FUNCTION_BLOCK "GCS7_M_Flift1Airlock"	// FB 66
TITLE = Fluidlift Blower with 1 Airlock
//  
//COPYRIGHT:    (C) 1997  BUHLER AG, CH-9240 UZWIL, SWITZERLAND
//
//PRODUCT:      GCS7
//
//TITLE:        FB 66 Machine Control:Fluidlift with 1 Airlock 
//              Blower, Blow off valve and Airlock
//
//-------------------------------------------------------------------------
//
//IDENT:        AUTHOR:             DEPT:                       DATE:
//
//FB66.4.2      A. Egli             CT3                         24-Nov-2004
//              Starting condition Airlock: Pressure.StMinP 
//FB66.4.1      A. Egli             CT3                         18-Aug-2003
//              No blow off, when Blower is started in manual mode 
//FB66.4.0      A. Egli             CT3                         17-Jun-2002
//              New Release with one block 
//FB66.3.4      A.Egli              CT3                         18-Mar-2002
//              Pressure.InLocal moved to segment "Global End"
//FB66.3.3      S. Kalberer         CT3                         23-Oct-2000
//              Blower stopped: Do not open BlowOff valve
//FB66.3.2      A. Egli             CT3                         25-Mai-2000
//              InNoWaitMinP 
//FB66.3.1      A. Egli             CT3                         2-Mai-2000
//              InMonMinP moved from segment "Interlocking" to "Gloabl End"
//FB66.3.0      A. Egli             CT3                         11-Oct-1999
//              Local data reduced
//FB66.2C       A. Egli             CT3                         27-Aug-1999
//              Interlocking Airlock with InEnable 
//FB66.2B       K. Tischer          MU664                       06-Mrz-1999
//              CC FC2 not UC FC2
//FB66.2A       A. Egli             CT3                         04-Mai-1998
//              StFault = StCode 32
//FB66.1A       A.Egli              AEE61                       5-Jul-1997
//              1st Release in S7
//
//-------------------------------------------------------------------------
//
//PURPOSE:      MANUAL : see [LL.FL1xxMAN]
//
//RESTRICTIONS: S7
//              ACCU2: Pointer to dynamic datas of the machine
//              ACCU1: Pointer to parameter datas of the machine
//
//-------------------------------------------------------------------------
//
AUTHOR : EA
FAMILY : GCS7LL
NAME : Fluid1
VERSION : 4.2
VAR
  Ma : UDT 20660;
  Pressure : FB 16;	//Element
  BlowOff : FB 13;	//Element
  Blower : FB 12;	//Element
  Airlock : FB 12;	//Element
  HLInlet : FB 14;	//Element
END_VAR
VAR_TEMP
  tmpFaultStop : BOOL ;
  tmpFaultSum : BOOL ;
  tmpBlowerStopped : BOOL ;
  tmpBlowerStarted : BOOL ;
  tmpBlowOffStLN : BOOL ;
  tmpLenDyn : INT ;
END_VAR
BEGIN
NETWORK
TITLE =
      L     18;
      T     #tmpLenDyn;
NETWORK
TITLE = PC Control
//=== Test Object number =====================
      L     "SYS_DirectCtrlDB".PC.ObjectNo;	//PCControl.ObjectNo
      L     #Ma.Par.ParObjectNo;	//Input ObjectNo
      <>I;
      JC    aEnd;
//=== Test OType      ========================
      L     2066;	//Input object type
      L     "SYS_DirectCtrlDB".PC.ObjectType;	//PCControl.ObjectType
      <>I;
      JC    aEnd;
//=== Test Handshake =========================
      A     "SYS_DirectCtrlDB".PC.Hsk.FExamine;	// Handshake.FExamine
      JC    aExa;
      A     "SYS_DirectCtrlDB".PC.Hsk.FDefineCmd;	// Handshake.FDefineCmd
      JC    aCmd;
      A     "SYS_DirectCtrlDB".PC.Hsk.FDefinePara;	// Handshake.FDefinePara
      JC    pPar;
aIni: L     2;	// FcInit
      UC    "SYS_DirectCtrl";
      JU    aEnd;
// Write parameter 
pPar: LAR1  P#DBX 58.0;
      L     P#6.0;
      +AR1;
      L     DBW [AR1,P#4.0];
      T     #Ma.Par.ParClearingTime;
// Write new commands from PC to Interface of group 
aCmd: A     "SYS_DirectCtrlDB".PC.Cmd1[8];	//Cmd1[8]=CmdOff
      S     #Ma.CmdOff;
      A     "SYS_DirectCtrlDB".PC.Cmd1[9];	//Cmd1[9]=CmdOn
      S     #Ma.CmdOn;
      A     "SYS_DirectCtrlDB".PC.Cmd1[10];	//Cmd1[10]=CmdNext
      S     #Ma.CmdNext;
      A     "SYS_DirectCtrlDB".PC.Cmd1[11];	//Cmd1[11]=CmdFaultReset
      S     #Ma.CmdFaultReset;
      A     "SYS_DirectCtrlDB".PC.Cmd1[13];	//Cmd1[13]=CmdManualOn
      S     #Ma.InManual;
      A     "SYS_DirectCtrlDB".PC.Cmd2[13];	//Cmd2[13]=CmdManualOff
      R     #Ma.InManual;
      A     "SYS_DirectCtrlDB".PC.Cmd1[14];	//Cmd1[14]=CmdManualOn
      S     #Ma.CmdAirlockOff;
      A     "SYS_DirectCtrlDB".PC.Cmd1[6];	//Cmd1[6]=CmdClearingOn
      S     #Ma.InClearing;
      A     "SYS_DirectCtrlDB".PC.Cmd2[6];	//Cmd2[6]=CmdClearingOff
      R     #Ma.InClearing;
      JU    aIni;
aExa: TAR2;	// Address Dynamic datas
      T     "SYS_DirectCtrlDB".GC.InDynAddr;	// -->PCControl.GC.InDynAddr
      L     #tmpLenDyn;	// Length Dynamic datas
      T     "SYS_DirectCtrlDB".GC.InDynLen;	// -->PCControl.GC.InDynLen
      L     0;
      T     "SYS_DirectCtrlDB".GC.InParaAddr;	// -->PCControl.GC.InParaAddr
      T     "SYS_DirectCtrlDB".GC.InParaLen;	// -->PCControl.GC.InParaLen
      L     1;	// Code FcExamine
      UC    "SYS_DirectCtrl";
      L     10;	//Revision
      T     "SYS_DirectCtrlDB".GC.Revision;
aEnd: NOP   0;
NETWORK
TITLE = Interlocking
//===Dynamic Group Orders===
      A     "GCS7_Gr_OutManualOn";	//Gr.OutManualOn
      S     #Ma.InManual;
      A     "GCS7_Gr_OutManualOff";	//Gr.OutManualOff
      R     #Ma.InManual;
      A     #Ma.InManual;
      S     "GCS7_Gr_InManual";	//Gr.InManual
//--- Fault----
      A     #Pressure.StFault;
      O     #BlowOff.StFault;
      O     #Blower.StFault;
      O     #Airlock.StFault;
      O     #HLInlet.StFault;
      =     #tmpFaultSum;
//Temporare signal
      A     #BlowOff.StLN;
      =     #tmpBlowOffStLN;
      A     #Ma.Par.ParBlowerExternal;
      A     #Ma.InBlowerStarted;
      O;
      AN    #Ma.Par.ParBlowerExternal;
      A     #Blower.StStartedFwd;
      =     #tmpBlowerStarted;
      A     #Ma.Par.ParBlowerExternal;
      AN    #Ma.InBlowerStarted;
      O;
      AN    #Ma.Par.ParBlowerExternal;
      A     #Blower.StStopped;
      =     #tmpBlowerStopped;
//--- Interlocking blow off
      A     #Ma.InClearing;
      A     #Ma.StCleared;
//[3.3]   ON    #tmpBlowerStarted;
      O     #Ma.InBlowOff;
      AN    #Blower.InManual;	//[4.1]
      =     #BlowOff.InEnableHN;
      AN    #BlowOff.InEnableHN;
      =     #BlowOff.InEnableLN;
//[->3.3  U     #Ma.CmdNext; 
//        UN    #Ma.InManual;
//        O     #Ma.CmdOn;
//        O     #tmpBlowerStarted;
      SET;	//<-3.3]
      S     #BlowOff.CmdNext;
// 
//--- Interlocking blower
      AN    #Pressure.StOverP;
      AN    #Pressure.StFault;
      =     #Ma.OutEnableBlower;
      AN    #Pressure.StOverP;
      AN    #Pressure.StFault;
      A     #Ma.InEnable;
      AN    #BlowOff.StFault;
      AN    #Ma.CmdOff;
      =     #Blower.InEnableFwd;
// 
//[3.3]   U     #BlowOff.StHN;
//[3.3]   ON    #Ma.Par.ParWithBlowOff;
//[3.3]   U(;
      A     #Ma.CmdNext;
      AN    #Ma.InManual;
      O     #Ma.CmdOn;
//[3.3]   ); 
      S     #Blower.CmdNext;
// 
      A     #Ma.InSeqStop;
      =     #Blower.InSeqStop;
// 
//--- Interlocking airlock 
      A     #BlowOff.StLN;
      ON    #Ma.Par.ParWithBlowOff;
      A     #tmpBlowerStarted;
      A     #Ma.InEnable;	// [Rel 2C]
      AN    #Ma.InClearing;
      AN    #Ma.InBlowOff;
      AN    #Pressure.StOverP;
      AN    #Pressure.StCtoOverP;
      AN    #Pressure.StFault;
      AN    #Ma.CmdOff;
      AN    #Ma.CmdAirlockOff;
      =     #Airlock.InEnableFwd;
// 
      A     #Ma.CmdNext;
      AN    #Ma.InManual;
      O     #Ma.CmdOn;
      A(;	//[4.2]
      A     #Pressure.StMinP;	//[4.2]
      O     #Ma.InNoWaitMinP;	//[4.2]
      );	//[4.2]
      S     #Airlock.CmdNext;
// 
      A     #Ma.InSeqStop;
      =     #Airlock.InSeqStop;
// 
//--- Local mode --
      A     #Ma.InLocal;
      AN    #Ma.InManual;
      =     #Blower.InLocal;
      =     #Airlock.InLocal;
      =     #HLInlet.InLocal;
      A     #Ma.InLocal;
      AN    #Ma.InManual;
      A     #tmpBlowerStopped;
      =     #BlowOff.InLocal;
//      =     #Pressure.InLocal //[3.4]
//--- Fault Reset -------------
      A     #Ma.CmdFaultReset;
      S     #Pressure.CmdFaultReset;
      S     #BlowOff.CmdFaultReset;
      S     #Blower.CmdFaultReset;
      S     #Airlock.CmdFaultReset;
      S     #HLInlet.CmdFaultReset;
//Warning
      A     #Pressure.OutNoMinP;
      =     #Ma.OutWarning;
NETWORK
TITLE = Call PRange: Pressure
      CALL  #Pressure;
NETWORK
TITLE = Call VLS: Blow off
      AN    #Ma.Par.ParWithBlowOff;
      JC    el3;
      CALL  #BlowOff;
NETWORK
TITLE = Call Blower
el3:  A     #Ma.Par.ParBlowerExternal;
      JC    el4;
      CALL  #Blower;
NETWORK
TITLE = Call Airlock
el4:  CALL  #Airlock;
NETWORK
TITLE = Call Digital Input: HLInlet
      AN    #Ma.Par.ParWithHLInlet;
      JC    StJ0;
      CALL  #HLInlet;
NETWORK
TITLE = Jump to actual state
StJ0: A     #Ma.StStopped;
      JC    S0;	// ===> State
      A     #Ma.StStarted;
      JC    S2;	// ===> State
      A     #Ma.StStarting;
      JC    S1;	// ===> State
      A     #Ma.StStopping;
      JC    S3;	// ===> State
      A     #Ma.StClearing;
      JC    S5;	// ===> State
      A     #Ma.StCleared;
      JC    S6;	// ===> State
      A     #Ma.StFault;
      JC    S4;	// ===> State
NETWORK
TITLE = Stopped
//any Transition 
xxS0: S     #Ma.StStopped;	// ===> Initialisation
//=== Logic
// Condition for StFault
S0:   A     #tmpFaultSum;
      R     #Ma.StStopped;
      JC    xxS4;	//--> StFault
// Condition for StStarting
      AN    #tmpBlowerStopped;
      ON    #Airlock.StStopped;
      R     #Ma.StStopped;
      JC    xxS1;	//--> StStarting
      JU    OUT;
NETWORK
TITLE = StStarting
//any Transition 
xxS1: S     #Ma.StStarting;
      JU    OUT;
//=== Logic
// Condition for StFault
S1:   A     #tmpFaultSum;
      R     #Ma.StStarting;
      JC    xxS4;	//--> StFault
// Condition for StStopping
      AN    #Blower.StStarting;
      AN    #Blower.StStartedFwd;
      AN    #tmpBlowerStarted;
      R     #Ma.StStarting;
      JC    xxS3;	//-->StStopping
// Condition for StStarted
      A     #BlowOff.StLN;
      ON    #Ma.Par.ParWithBlowOff;
      A     #tmpBlowerStarted;
      A     #Airlock.StStartedFwd;
      R     #Ma.StStarting;
      JC    xxS2;	//-->StStarted
// Condition for StClearing
      AN    #Ma.Par.ParWithBlowOff;
      O     #tmpBlowOffStLN;
      A     #tmpBlowerStarted;
      AN    #Airlock.StStarting;
      R     #Ma.StStarting;
      JC    xxS5;	//-->StClearing
      JU    OUT;
NETWORK
TITLE = StStarted
//any Transition 
xxS2: S     #Ma.StStarted;
//=== Logic
// Condition for StFault
S2:   A     #tmpFaultSum;
      R     #Ma.StStarted;
      JC    xxS4;	//--> StFault
// Condition for StClearing
      AN    #Airlock.StStartedFwd;
      R     #Ma.StStarted;
      JC    xxS5;	//-->StClearing  
// Condition for StStarted
      ON    #tmpBlowerStarted;
      R     #Ma.StStarted;
      JC    xxS3;	//-->StStopping
      JU    OUT;
NETWORK
TITLE = Stopping
//any Transition 
xxS3: S     #Ma.StStopping;
      JU    OUT;
//=== Logic
// Condition for StFault
S3:   A     #tmpFaultSum;
      R     #Ma.StStopping;
      JC    xxS4;	//--> StFault
// Condition for StStopped
      A     #tmpBlowerStopped;
      A     #Airlock.StStopped;
      R     #Ma.StStopping;
      JC    xxS0;	//-->StStopped
// Condition for StStarting
      AN    #Blower.StStopping;
      AN    #Ma.Par.ParBlowerExternal;
      O     #tmpBlowerStarted;
      AN    #Airlock.StStopping;
      R     #Ma.StStopping;
      JC    xxS1;	//-->StStarting
      JU    OUT;
NETWORK
TITLE = Fault
//any Transition 
xxS4: S     #Ma.StFault;
      JU    OUT;
//=== Logic
S4:   A     #tmpFaultSum;
      JC    OUT;
//    ---- Transition --
      R     #Ma.StFault;
      JU    xxS0;	//-->StStopping 
NETWORK
TITLE = StClearing
//any Transition 
xxS5: S     #Ma.StClearing;
S5J2: L     #Ma.Par.ParClearingTime;
      T     #Ma.Par.OutClearingTime;
      JU    OUT;
//=== Logic
// Condition for StFault
S5:   A     #tmpFaultSum;
      R     #Ma.StClearing;
      JC    xxS4;	//-->StFault
// Condition for StStopping
      AN    #tmpBlowerStarted;
      R     #Ma.StClearing;
      JC    xxS3;	//-->StStopping  
// Condition for StStarted
      A     #tmpBlowerStarted;
      A     #Airlock.StStartedFwd;
      R     #Ma.StClearing;
      JC    xxS2;	//-->StStarted
// Condition for StCleared
      L     0;
      L     #Ma.Par.OutClearingTime;
      >=I;
      A(;
      A     #Pressure.StMinP;
      O     #Ma.InNoWaitMinP;	// [3.2]
      );
      R     #Ma.StClearing;
      JC    xxS6;	//-->StCleared 
      AN    #BlowOff.StLN;
      A     #Ma.Par.ParWithBlowOff;
      O;
      AN    #Pressure.StMinP;
      AN    #Ma.InNoWaitMinP;	// [3.2]
      JC    S5J2;
      ON    "GCS7_Gr_OutTick500ms";	//Gr.OutTick500ms
      JC    OUT;
      +     -5;
      T     #Ma.Par.OutClearingTime;
      JU    OUT;
NETWORK
TITLE = StCleared
//any Transition 
xxS6: S     #Ma.StCleared;
      JU    OUT;
//=== Logic
// Condition for StFault
S6:   A     #tmpFaultSum;
      R     #Ma.StCleared;
      JC    xxS4;	//-->StFault
// Condition for StStopping
      AN    #tmpBlowerStarted;
      R     #Ma.StCleared;
      JC    xxS3;	//-->StStopping
// Condition for StStarted
      A     #tmpBlowerStarted;
      A     #Airlock.StStartedFwd;
      R     #Ma.StCleared;
      JC    xxS2;	//-->StStarted
      JU    OUT;
NETWORK
TITLE = State Code
// State     StCode
// ----------------------
// StFault 32
// StStopped          1
// StStarting         2
// StStarted          3
// StClearing         4
// StCleared          5
// StClearingWarning  6
// StStopping         7
OUT:  A     #Ma.StStopped;
      L     1;	//Code=StStopped
      JC    Code;
      A     #Ma.StStarted;
      L     3;	//Code=StStarted
      JC    Code;
      A     #Ma.StCleared;
      L     5;	//Code=StCleared
      JC    Code;
      A     #Ma.StClearing;
      AN    #Ma.OutWarning;
      L     4;	//Code=StClearing 
      JC    Code;
      A     #Ma.StClearing;
      L     6;	//Code=StWarning 
      JC    Code;
      A     #Ma.StStarting;
      L     2;	//Code=StStarting
      JC    Code;
      A     #Ma.StStopping;
      L     7;	//Code=StStopping 
      JC    Code;
      L     32;	//Code=StFault 
Code: L     #Ma.StCode;	// Old state code
      TAK;
      T     #Ma.StCode;	// Save state code
      <>I;
      L     3;
      CC    "SYS_CBitCtrl";	//Set change bit
NETWORK
TITLE = Global End
      CLR;	//---Clear all commands
      =     #Ma.CmdOn;
      =     #Ma.CmdOff;
      =     #Ma.CmdNext;
      =     #Ma.CmdFaultReset;
      =     #Ma.CmdAirlockOff;
// 
//--- Interlocking pressure 
      A     #BlowOff.StLN;
      ON    #Ma.Par.ParWithBlowOff;
      AN    #Airlock.StStartedFwd;
      A     #tmpBlowerStarted;
      =     #Pressure.InMonMinP;
// 
//--- Local mode --       
      A     #BlowOff.InLocal;	//[3.4]
      =     #Pressure.InLocal;	//[3.4]
// 
//--- Interlocking HL 
      SET;
      =     #HLInlet.InMonFalse;
END_FUNCTION_BLOCK

FUNCTION_BLOCK "GCS7_M_Flift2Airlock"	// FB 67
TITLE = Fluidlift Blower with 2 Airlock
//  
//COPYRIGHT:    (C) 1997  BUHLER AG, CH-9240 UZWIL, SWITZERLAND
//
//PRODUCT:      GCS7
//
//TITLE:        FB 67 Machine Control:Fluidlift 2 Airlock and 2 Shutoff Valve
//              Blower, Blow off valve and Airlock
//
//-------------------------------------------------------------------------
//
//IDENT:        AUTHOR:             DEPT:                       DATE:
//
//FB67.6.7      A. Egli             BASE                        10-Apr-2008
//              StStarting -> StStopping ParExternal
//FB67.6.6      A. Egli             CT3                         04-Mar-2005
//              Support continuous valve for ShutOff and BlowOff 
//FB67.6.5      A. Egli             CT3                         04-Mar-2005
//              Start Blower before opening ShutOffA or ShutOffB 
//FB67.6.4      A. Egli             CT3                         20-Sep-2004
//              Interlocking Subtype Diverter without BlowOff valve
//FB67.6.3      A. Egli             CT3                         10-Jun-2004
//              Diverter.InLocal
//FB67.6.2      A. Egli             CT3                         19-Sep-2003
//              InMonFalse mode to global end function
//FB67.6.1      A. Egli             CT3                         18-Aug-2003
//              No blow off, when Blower is started in manual mode 
//FB67.6.0      A. Egli             CT3                         17-Jun-2002
//              New Release with one block 
//FB67.5.7      A.Egli              CT3                         18-Mar-2002
//              Pressure.InLocal moved to segment "Global End"
//FB67.5.6      A.Egli              CT3                         29-Oct-2001
//              InLocal of HL moved to segment "Global End"
//FB67.5.5      A.Egli              CT3                         16-May-2001
//              - Close Valve with InSeqStop
//              - Monitoring only active HLInlet  
//FB67.5.4      Ph.Engler           MU664                       15-May-2001
//              - Diverter.CmdFaultReset corrected
//FB67.5.3      Ph.Engler           MU664                       08-Jan-2000
//              InBlowOff without a blowoff valve closes directly
//              the ShutOffA valve.
//FB67.5.2      Ph.Engler           MU664                       29-Dec-2000
//              - Enable airlock A on a single line type and shutt off valve
//              - OutEnableBlower implemented
//              - InMonMinP moved from segment "Interlocking" to "Gloabl End"
//FB67.5.1      S. Kalberer         CT3                         23-Oct-2000
//              Blower stopped: Do not open BlowOff valve
//FB67.5.0      A. Egli             CT3                    20-Sep-2000
//              With Diverter valve
//FB67.4.0      A. Egli             CT3                    26-Mai-2000
//              Single line with ShutOff valves
//              InNoWaitMinP 
//FB67.3.1      A. Egli             CT3                    28-Jan-2000
//              Interlocking blower
//FB67.3.0      A. Egli             CT3                         11-Oct-1999
//              Local data reduced
//FB67.2B       K. Tischer          MU664                       06-Mrz-1999
//              CC FC2 not UC FC2
//FB67.2A       A. Egli             CT3                         04-Mai-1998
//              StFault = StCode 32
//FB67.1A       A. Egli              AEE61                      27-Nov-1997
//              1st Release in S7
//
//-------------------------------------------------------------------------
//
//PURPOSE:      MANUAL : see [LL.FL2xxMAN]
//
//RESTRICTIONS: S7
//              ACCU2: Pointer to dynamic datas of the machine
//              ACCU1: Pointer to parameter datas of the machine
//
//-------------------------------------------------------------------------
//
AUTHOR : EA
FAMILY : GCS7LL
NAME : Fluid2AV
VERSION : 6.6
VAR
  Ma : UDT 20670;
  Pressure : FB 16;	//Element
  BlowOff : FB 13;	//Element
  Blower : FB 12;	//Element
  ShutOffA : FB 13;	//Element
  ShutOffB : FB 13;	//Element
  AirlockA : FB 12;	//Element
  AirlockB : FB 12;	//Element
  HLInletA : FB 14;	//Element
  HLInletB : FB 14;	//Element
  Diverter : FB 13;	//Element
END_VAR
VAR_TEMP
  tmpFaultStop : BOOL ;
  tmpFaultSum : BOOL ;
  tmpEnable : BOOL ;
  tmpEnableAirlock : BOOL ;
  tmpNext : BOOL ;
  tmpBlowOff : BOOL ;
  tmpBlowerStopped : BOOL ;
  tmpBlowerStarted : BOOL ;
  tmpBlowOffStLN : BOOL ;
  tmpWayA : BOOL ;
  tmpWayB : BOOL ;
  tmpWithShutOffValves : BOOL ;
  tmpWithDiverterValves : BOOL ;
  tmpWayAOK : BOOL ;
  tmpWayBOK : BOOL ;
  tmpCloseValve : BOOL ;
  tmpPressureLocal : BOOL ;
  tmpLenDyn : INT ;
END_VAR
BEGIN
NETWORK
TITLE =
      L     18;
      T     #tmpLenDyn;
NETWORK
TITLE = PC Control
//=== Test Object number =====================
      L     "SYS_DirectCtrlDB".PC.ObjectNo;	//PCControl.ObjectNo
      L     #Ma.Par.ParObjectNo;	//Input ObjectNo
      <>I;
      JC    aEnd;
//=== Test OType  ========================
      L     2067;	//Input object type
      L     "SYS_DirectCtrlDB".PC.ObjectType;	//PCControl.ObjectType
      <>I;
      JC    aEnd;
//=== Test Handshake =========================
      A     "SYS_DirectCtrlDB".PC.Hsk.FExamine;	// Handshake.FExamine
      JC    aExa;
      A     "SYS_DirectCtrlDB".PC.Hsk.FDefineCmd;	// Handshake.FDefineCmd
      JC    aCmd;
      A     "SYS_DirectCtrlDB".PC.Hsk.FDefinePara;	// Handshake.FDefinePara
      JC    pPar;
aIni: L     2;	// FcInit
      UC    "SYS_DirectCtrl";
      JU    aEnd;
// Write parameter 
pPar: LAR1  P#DBX 58.0;
      L     P#6.0;
      +AR1;
      L     DBW [AR1,P#4.0];
      T     #Ma.Par.ParClearingTime;
// Write new commands from PC to Interface of group 
aCmd: A     "SYS_DirectCtrlDB".PC.Cmd1[8];	//Cmd1[8]=CmdOff
      S     #Ma.CmdOff;
      A     "SYS_DirectCtrlDB".PC.Cmd1[9];	//Cmd1[9]=CmdOn
      S     #Ma.CmdOn;
      A     "SYS_DirectCtrlDB".PC.Cmd1[10];	//Cmd1[10]=CmdNext
      S     #Ma.CmdNext;
      A     "SYS_DirectCtrlDB".PC.Cmd1[11];	//Cmd1[11]=CmdFaultReset
      S     #Ma.CmdFaultReset;
      A     "SYS_DirectCtrlDB".PC.Cmd1[13];	//Cmd1[13]=CmdManualOn
      S     #Ma.InManual;
      A     "SYS_DirectCtrlDB".PC.Cmd2[13];	//Cmd2[13]=CmdManualOff
      R     #Ma.InManual;
      A     "SYS_DirectCtrlDB".PC.Cmd1[14];	//Cmd1[14]=CmdManualOn
      S     #Ma.CmdAirlockOff;
      A     "SYS_DirectCtrlDB".PC.Cmd1[1];	//Cmd1[1]=CmdWayA
      R     #Ma.InWayB;
      A     "SYS_DirectCtrlDB".PC.Cmd2[1];	//Cmd2[2]=CmdWayB
      S     #Ma.InWayB;
      A     "SYS_DirectCtrlDB".PC.Cmd1[6];	//Cmd1[6]=CmdClearingOn
      S     #Ma.InClearing;
      A     "SYS_DirectCtrlDB".PC.Cmd2[6];	//Cmd2[6]=CmdClearingOff
      R     #Ma.InClearing;
      JU    aIni;
aExa: TAR2;	// Address Dynamic datas
      T     "SYS_DirectCtrlDB".GC.InDynAddr;	// -->PCControl.GC.InDynAddr
      L     #tmpLenDyn;	// Length Dynamic datas
      T     "SYS_DirectCtrlDB".GC.InDynLen;	// -->PCControl.GC.InDynLen
      L     0;
      T     "SYS_DirectCtrlDB".GC.InParaAddr;	// -->PCControl.GC.InParaAddr
      T     "SYS_DirectCtrlDB".GC.InParaLen;	// -->PCControl.GC.InParaLen
      L     1;	// Code FcExamine
      UC    "SYS_DirectCtrl";
      L     10;	//Revision
      T     "SYS_DirectCtrlDB".GC.Revision;
aEnd: NOP   0;
NETWORK
TITLE = Interlocking
//===Dynamic Group Orders===
      A     "GCS7_Gr_OutManualOn";	//Gr.OutManualOn
      S     #Ma.InManual;
      A     "GCS7_Gr_OutManualOff";	//Gr.OutManualOff
      R     #Ma.InManual;
      A     #Ma.InManual;
      S     "GCS7_Gr_InManual";	//Gr.InManual
      A     #Ma.InManual;
      ON    #Ma.InLocal;
      A     #Ma.InEnable;
      AN    #Ma.CmdOff;
      =     #tmpEnable;
//Temporare signal
      AN    #Ma.InWayB;
      O     #Ma.InWayAB;
      =     #tmpWayA;
      A     #Ma.InWayB;
      O     #Ma.InWayAB;
      =     #tmpWayB;
      A     #BlowOff.StLN;
      =     #tmpBlowOffStLN;
      A     #Ma.Par.ParWithShutOffValves;
      ON    #Ma.Par.ParSingleLine;
      =     #tmpWithShutOffValves;
      A     #Ma.Par.ParBlowerExternal;
      A     #Ma.InBlowerStarted;
      O;
      AN    #Ma.Par.ParBlowerExternal;
      A     #Blower.StStartedFwd;
      =     #tmpBlowerStarted;
      A     #Ma.Par.ParBlowerExternal;
      AN    #Ma.InBlowerStarted;
      O;
      AN    #Ma.Par.ParBlowerExternal;
      A     #Blower.StStopped;
      =     #tmpBlowerStopped;
      A     #Ma.InSeqStop;	//[5.5]
      O     #Ma.InLocal;	//[5.5]
      AN    #Ma.InManual;	//[5.5]
      A     #tmpBlowerStopped;	//[5.5]
      AN    #Blower.InManual;	//[6.1]
      =     #tmpCloseValve;	//[5.5]
//--- Fault----
      A     #Diverter.StFault;
      A     #Ma.Par.ParWithDiverter;
      O     #Pressure.StFault;
      O     #BlowOff.StFault;
      O     #ShutOffA.StFault;
      O     #ShutOffB.StFault;
      O     #Blower.StFault;
      O     #AirlockA.StFault;
      O     #AirlockB.StFault;
      O     #HLInletA.StFault;
      O     #HLInletB.StFault;
      =     #tmpFaultSum;
//CmdNext
      A     #Ma.CmdNext;
      AN    #Ma.InManual;
      O     #Ma.CmdOn;
      =     #tmpNext;
//[5.1]   U       #BlowOff.StHN;
//[5.1]   ON      #Ma.Par.ParWithBlowOff;
      A     #tmpNext;
      S     #Blower.CmdNext;
      A     #tmpNext;
      S     #Blower.CmdNext;
      S     #AirlockA.CmdNext;
      S     #AirlockB.CmdNext;
      SET;
      S     #BlowOff.CmdNext;
      A(;	//[6.5]
      A     #tmpBlowerStarted;	//[6.5]
      ON    #Ma.Par.ParWithBlowOff;	//[6.5]
      );	//[6.5]
      O;
      A     #ShutOffA.InEnableLN;	//[6.5]
      AN    #ShutOffA.StLN;	//[6.5]
      S     #ShutOffA.CmdNext;
      A(;	//[6.5]
      A     #tmpBlowerStarted;	//[6.5]
      ON    #Ma.Par.ParWithBlowOff;	//[6.5]
      );	//[6.5]
      O(;
      A     #ShutOffB.InEnableLN;	//[6.5]
      AN    #ShutOffB.StLN;	//[6.5]
      );
      S     #ShutOffB.CmdNext;
      AN    #Ma.Par.ParWithDiverter;
      JC    InX1;
      S     #Diverter.CmdNext;
//--- Interlocking blow off
InX1: A     #Diverter.StLN;
      ON    #Ma.Par.ParWithDiverter;
      A     #ShutOffA.StHN;
      A(;
      A     #tmpWayA;
      O     #Ma.Par.ParSingleLine;
      );
      =     #tmpWayAOK;
      A     #Diverter.StHN;
      ON    #Ma.Par.ParWithDiverter;
      A     #ShutOffB.StHN;
      A     #tmpWayB;
      AN    #Ma.Par.ParSingleLine;
      =     #tmpWayBOK;
      A     #Ma.InClearing;
      A     #Ma.StCleared;
//[5.1]   ON      #tmpBlowerStarted;
      O     #Ma.InBlowOff;
      A     #Ma.Par.ParWithBlowOff;
      =     #tmpBlowOff;
      AN    #tmpWayAOK;
      AN    #tmpWayBOK;
      A     #tmpWithShutOffValves;
      O     #tmpBlowOff;
      AN    #tmpCloseValve;	//[5.5]
      =     #BlowOff.InEnableHN;
      AN    #BlowOff.InEnableHN;
      =     #BlowOff.InEnableLN;
//--- Interlocking ShutOff Valve
      A     #Diverter.StHN;	//[6.4]
      ON    #Ma.Par.ParWithDiverter;	//[6.4]
      A     #ShutOffB.StHN;
      A     #tmpWayB;
      AN    #tmpWayA;
      O;
      A     #tmpBlowOff;
      A     #BlowOff.StHN;
      O;
      A     #Ma.InBlowOff;
      AN    #Ma.Par.ParWithBlowOff;
      O;
      A     #BlowOff.StHN;
      A     #tmpWayB;
      A     #Ma.Par.ParWithDiverter;
      O     #tmpCloseValve;	//[5.5]
      =     #ShutOffA.InEnableLN;
      R     #ShutOffA.InEnableHN;	//[6.6]
      A     #tmpWayA;
      O     #Ma.Par.ParSingleLine;
      AN    #ShutOffA.InEnableLN;
      A(;
      A     #ShutOffB.StHN;	//[6.4]
      AN    #Ma.Par.ParWithBlowOff;	//[6.4]
      O     #Diverter.StLN;
      ON    #Ma.Par.ParWithDiverter;
      );
      S     #ShutOffA.InEnableHN;	//[6.6]
      R     #ShutOffA.InEnableLN;	//[6.6]
      A     #Diverter.StLN;	//[6.4]
      ON    #Ma.Par.ParWithDiverter;	//[6.4]
      A     #ShutOffA.StHN;
      A     #tmpWayA;
      AN    #tmpWayB;
      O;
      A     #tmpBlowOff;
      A     #BlowOff.StHN;
      O;
      A     #BlowOff.StHN;
      A     #tmpWayA;
      A     #Ma.Par.ParWithDiverter;
      O     #tmpCloseValve;	//[5.5]
      =     #ShutOffB.InEnableLN;
      R     #ShutOffB.InEnableHN;	//[6.6]
      AN    #ShutOffB.InEnableLN;
      A     #tmpWayB;
      A(;
      A     #ShutOffA.StHN;	//[6.4]
      AN    #Ma.Par.ParWithBlowOff;	//[6.4]
      O     #Diverter.StHN;
      ON    #Ma.Par.ParWithDiverter;
      );
      S     #ShutOffB.InEnableHN;	//[6.6]
      R     #ShutOffB.InEnableLN;	//[6.6]
//--- Interlocking blower
      AN    #Pressure.StOverP;	//[5.2]
      AN    #Pressure.StFault;	//[5.2]
      =     #Ma.OutEnableBlower;	//[5.2]
      A     #BlowOff.StHN;
      A     #Ma.Par.ParWithBlowOff;
      O     #ShutOffA.StHN;	//[3.1]
      O     #ShutOffB.StHN;	//[3.1]
      ON    #tmpWithShutOffValves;	//[4.0]
      A     #tmpEnable;
      AN    #Pressure.StOverP;
      AN    #Pressure.StFault;
      AN    #BlowOff.StFault;
      =     #Blower.InEnableFwd;
// 
      A     #Ma.InSeqStop;
      AN    #Ma.InManual;	//[5.5]
      =     #Blower.InSeqStop;
// 
//--- Interlocking airlock 
      A     #BlowOff.StLN;
      ON    #Ma.Par.ParWithBlowOff;
      AN    #Ma.InClearing;
      A     #tmpEnable;
      A     #tmpBlowerStarted;
      AN    #Pressure.StOverP;
      AN    #Pressure.StCtoOverP;
      AN    #Pressure.StFault;
      AN    #Ma.CmdAirlockOff;
      AN    #Ma.InBlowOff;
      =     #tmpEnableAirlock;
      A     #ShutOffB.StLN;
      O     #tmpWayB;
      O     #Ma.Par.ParSingleLine;	//[5.2]
      A     #ShutOffA.StHN;
      ON    #tmpWithShutOffValves;
      A     #tmpEnableAirlock;
      A     #tmpWayA;
      AN    #Ma.InDisableAirlockA;
      A(;
      A     #Diverter.StLN;
      ON    #Ma.Par.ParWithDiverter;
      );
      =     #AirlockA.InEnableFwd;
      A     #ShutOffA.StLN;
      O     #tmpWayA;
      A     #ShutOffB.StHN;
      A     #tmpEnableAirlock;
      A     #tmpWayB;
      AN    #Ma.Par.ParSingleLine;
      O(;
      A     #ShutOffA.StHN;
      ON    #tmpWithShutOffValves;
      A     #tmpEnableAirlock;
      A     #tmpWayB;
      O     #AirlockA.InEnableFwd;
      A     #Ma.Par.ParSingleLine;
      );
      AN    #Ma.InDisableAirlockB;
      A(;
      A     #Diverter.StHN;
      ON    #Ma.Par.ParWithDiverter;
      );
      =     #AirlockB.InEnableFwd;
// 
      A     #Ma.InSeqStop;
      AN    #Ma.InManual;	//[5.5]
      =     #AirlockA.InSeqStop;
      =     #AirlockB.InSeqStop;
// 
//--- Interlocking pressure  [5.2] moved to "global end"
// 
//--- Interlocking HL        [6.2] moved to "global end"
//--- Interlocking Diverter
      AN    #Ma.Par.ParWithDiverter;
      JC    EnX1;
      A(;	//[6.4]
      A     #BlowOff.StHN;
      A     #ShutOffB.StLN;	//[6.4]
      A     #Ma.Par.ParWithBlowOff;	//[6.4]
      O;
      A     #ShutOffA.StHN;	//[6.4]
      AN    #Ma.Par.ParWithBlowOff;	//[6.4]
      O;
      A     #ShutOffB.StLN;	//[6.4]
      AN    #Ma.Par.ParWithBlowOff;	//[6.4]
      );	//[6.4]
      A     #tmpWayA;
      S     #Diverter.InEnableLN;
      R     #Diverter.InEnableHN;
      A(;	//[6.4]
      A     #BlowOff.StHN;
      A     #ShutOffA.StLN;	//[6.4]
      A     #Ma.Par.ParWithBlowOff;	//[6.4]
      O;
      A     #ShutOffB.StHN;	//[6.4]
      AN    #Ma.Par.ParWithBlowOff;	//[6.4]
      O;
      A     #ShutOffA.StLN;	//[6.4]
      AN    #Ma.Par.ParWithBlowOff;	//[6.4]
      );	//[6.4]
      A     #tmpWayB;
      R     #Diverter.InEnableLN;
      S     #Diverter.InEnableHN;
// 
//--- Local mode --
EnX1: A     #Ma.InLocal;
      AN    #Ma.InManual;
      =     #Blower.InLocal;
      =     #AirlockA.InLocal;
      =     #AirlockB.InLocal;
      =     #Diverter.InLocal;	//[6.3]
      A     #Ma.InLocal;
      AN    #Ma.InManual;
      A     #tmpBlowerStopped;
      =     #tmpPressureLocal;
      A     #BlowOff.StLN;	//[5.5]
      O     #BlowOff.StFault;	//[5.5]
      A     #tmpPressureLocal;	//[5.5]
      S     #BlowOff.InLocal;	//[5.5]
      A     #ShutOffA.StLN;	//[5.5]
      O     #ShutOffA.StFault;	//[5.5]
      A     #tmpPressureLocal;	//[5.5]
      S     #ShutOffA.InLocal;	//[5.5]
      A     #ShutOffB.StLN;	//[5.5]
      O     #ShutOffB.StFault;	//[5.5]
      A     #tmpPressureLocal;	//[5.5]
      S     #ShutOffB.InLocal;	//[5.5]
      AN    #tmpPressureLocal;	//[5.5]
      R     #BlowOff.InLocal;
      R     #ShutOffA.InLocal;
      R     #ShutOffB.InLocal;
//--- Fault Reset -------------
      A     #Ma.CmdFaultReset;
      S     #Pressure.CmdFaultReset;
      S     #BlowOff.CmdFaultReset;
      S     #ShutOffA.CmdFaultReset;
      S     #ShutOffB.CmdFaultReset;
      S     #Blower.CmdFaultReset;
      S     #AirlockA.CmdFaultReset;
      S     #AirlockB.CmdFaultReset;
      S     #HLInletA.CmdFaultReset;
      S     #HLInletB.CmdFaultReset;
      AN    #Ma.Par.ParWithDiverter;
      JC    FrX1;
      A     #Ma.CmdFaultReset;	// [5.4]
      S     #Diverter.CmdFaultReset;
//Warning
FrX1: A     #Pressure.OutNoMinP;
      =     #Ma.OutWarning;
NETWORK
TITLE = Call PRange: Pressure
      CALL  #Pressure;
NETWORK
TITLE = Call VLS: Blow off
      AN    #Ma.Par.ParWithBlowOff;
      JC    el3;
      CALL  #BlowOff;
NETWORK
TITLE = Call VLS: ShutOffA
el3:  AN    #tmpWithShutOffValves;
      JC    el4;
      CALL  #ShutOffA;
NETWORK
TITLE = Call VLS: ShutOffB
el4:  A     #Ma.Par.ParSingleLine;
      JC    el5;
      CALL  #ShutOffB;
NETWORK
TITLE = Call Blower
el5:  A     #Ma.Par.ParBlowerExternal;
      JC    el6;
      CALL  #Blower;
NETWORK
TITLE = Call AirlockA
el6:  CALL  #AirlockA;
NETWORK
TITLE = Call AirlockB
      CALL  #AirlockB;
NETWORK
TITLE = Call Digital Input: HLInletA
      CALL  #HLInletA;
NETWORK
TITLE = Call Digital Input: HLInletB
      CALL  #HLInletB;
NETWORK
TITLE = Call Digital Output: Diverter
      AN    #Ma.Par.ParWithDiverter;
      JC    SPen;
      CALL  #Diverter;
SPen: NOP   0;
NETWORK
TITLE = Jump to actual state
      A     #Ma.StStopped;
      JC    S0;	// ===> State
      A     #Ma.StStarted;
      JC    S2;	// ===> State
      A     #Ma.StStarting;
      JC    S1;	// ===> State
      A     #Ma.StStopping;
      JC    S3;	// ===> State
      A     #Ma.StClearing;
      JC    S5;	// ===> State
      A     #Ma.StCleared;
      JC    S6;	// ===> State
      A     #Ma.StFault;
      JC    S4;	// ===> State
NETWORK
TITLE = Stopped
//any Transition 
xxS0: S     #Ma.StStopped;	// ===> Initialisation
      JU    OUT;
//=== Logic
// Condition for StFault
S0:   A     #tmpFaultSum;
      R     #Ma.StStopped;
      JC    xxS4;	//--> ST_FAULT:
// Condition for StStarting
      AN    #tmpBlowerStopped;
      ON    #AirlockA.StStopped;
      ON    #AirlockB.StStopped;
      R     #Ma.StStopped;
      JC    xxS1;	//--> StStarting
      JU    OUT;
NETWORK
TITLE = StStarting
//any Transition 
xxS1: S     #Ma.StStarting;
      JU    OUT;
//=== Logic
// Condition for StFault
S1:   A     #tmpFaultSum;
      R     #Ma.StStarting;
      JC    xxS4;	//--> StFault
// Condition for StStopping
      AN    #Blower.StStarting;
      O     #Ma.Par.ParBlowerExternal;	//[6.7]
      AN    #tmpBlowerStarted;
      R     #Ma.StStarting;
      JC    xxS3;	//-->StStopping
// Condition for StStarted
      A     #AirlockA.StStartedFwd;
      O     #AirlockB.StStartedFwd;
      A     #tmpBlowerStarted;
      R     #Ma.StStarting;
      JC    xxS2;	//-->StStarted
// Condition for StClearing
      AN    #Ma.Par.ParWithBlowOff;
      O     #tmpBlowOffStLN;
      A     #tmpBlowerStarted;
      AN    #AirlockA.StStarting;
      AN    #AirlockB.StStarting;
      R     #Ma.StStarting;
      JC    xxS5;	//-->StClearing
      JU    OUT;
NETWORK
TITLE = StStarted
//any Transition 
xxS2: S     #Ma.StStarted;
      JU    OUT;
//=== Logic
// Condition for StFault
S2:   A     #tmpFaultSum;
      R     #Ma.StStarted;
      JC    xxS4;	//--> StFault
// Condition for StClearing
      AN    #AirlockA.StStartedFwd;
      AN    #AirlockB.StStartedFwd;
      R     #Ma.StStarted;
      JC    xxS5;	//-->StClearing  
// Condition for StStarted
      AN    #tmpBlowerStarted;
      R     #Ma.StStarted;
      JC    xxS3;	//-->StStopping
      JU    OUT;
NETWORK
TITLE = Stopping
//any Transition 
xxS3: S     #Ma.StStopping;
      JU    OUT;
//=== Logic
// Condition for StFault
S3:   A     #tmpFaultSum;
      R     #Ma.StStopping;
      JC    xxS4;	//--> StFault
// Condition for StStopped
      A     #tmpBlowerStopped;
      A     #AirlockA.StStopped;
      A     #AirlockB.StStopped;
      R     #Ma.StStopping;
      JC    xxS0;	//-->StStopped
// Condition for StStarting
      AN    #Blower.StStopping;
      AN    #Ma.Par.ParBlowerExternal;
      O     #tmpBlowerStarted;
      AN    #AirlockA.StStopping;
      AN    #AirlockB.StStopping;
      R     #Ma.StStopping;
      JC    xxS1;	//-->StStarting
      JU    OUT;
NETWORK
TITLE = Fault
//any Transition 
xxS4: S     #Ma.StFault;
      JU    OUT;
//=== Logic
S4:   A     #tmpFaultSum;
      JC    OUT;
//    ---- Transition --
      R     #Ma.StFault;
      JU    xxS0;	//-->StStopping 
NETWORK
TITLE = StClearing
//any Transition 
xxS5: S     #Ma.StClearing;
S5J2: L     #Ma.Par.ParClearingTime;
      T     #Ma.Par.OutClearingTime;
      JU    OUT;
//=== Logic
// Condition for StFault
S5:   A     #tmpFaultSum;
      R     #Ma.StClearing;
      JC    xxS4;	//-->StFault
// Condition for StStopping
      AN    #tmpBlowerStarted;
      R     #Ma.StClearing;
      JC    xxS3;	//-->StStopping  
// Condition for StStarted
      A     #AirlockA.StStartedFwd;
      O     #AirlockB.StStartedFwd;
      A     #tmpBlowerStarted;
      R     #Ma.StClearing;
      JC    xxS2;	//-->StStarted
// Condition for StCleared
      L     0;
      L     #Ma.Par.OutClearingTime;
      >=I;
      A(;
      A     #Pressure.StMinP;
      O     #Ma.InNoWaitMinP;	// [4.0]
      );
      R     #Ma.StClearing;
      JC    xxS6;	//-->StCleared 
      AN    #BlowOff.StLN;
      A     #Ma.Par.ParWithBlowOff;
      O;
      AN    #Pressure.StMinP;
      AN    #Ma.InNoWaitMinP;	// [4.0]
      JC    S5J2;
      ON    "GCS7_Gr_OutTick500ms";	//Gr.OutTick500ms
      JC    OUT;
      +     -5;
      T     #Ma.Par.OutClearingTime;
      JU    OUT;
NETWORK
TITLE = StCleared
//any Transition 
xxS6: S     #Ma.StCleared;
      JU    OUT;
//=== Logic
// Condition for StFault
S6:   A     #tmpFaultSum;
      R     #Ma.StCleared;
      JC    xxS4;	//-->StFault
// Condition for StStopping
      AN    #tmpBlowerStarted;
      R     #Ma.StCleared;
      JC    xxS3;	//-->StStopping
// Condition for StStarted
      A     #AirlockA.StStartedFwd;
      O     #AirlockB.StStartedFwd;
      A     #tmpBlowerStarted;
      R     #Ma.StCleared;
      JC    xxS2;	//-->StStarted
      JU    OUT;
NETWORK
TITLE = State Code
// State     StCode
// ----------------------
// StFault32
// StStopped    1
// StStarting   2
// StStarted    3
// StClearing   4
// StCleared    5
// StClearingWarning  6
// StStopping   7
OUT:  A     #Ma.StStopped;
      L     1;	//Code=StStopped
      JC    Code;
      A     #Ma.StStarted;
      L     3;	//Code=StStarted
      JC    Code;
      A     #Ma.StCleared;
      L     5;	//Code=StCleared
      JC    Code;
      A     #Ma.StClearing;
      AN    #Ma.OutWarning;
      L     4;	//Code=StClearing 
      JC    Code;
      A     #Ma.StClearing;
      L     6;	//Code=StWarning 
      JC    Code;
      A     #Ma.StStarting;
      L     2;	//Code=StStarting
      JC    Code;
      A     #Ma.StStopping;
      L     7;	//Code=StStopping 
      JC    Code;
      L     32;	//Code=StFault 
Code: L     #Ma.StCode;	// Old state code
      TAK;
      T     #Ma.StCode;	// Save state code
      <>I;
      L     3;
      CC    "SYS_CBitCtrl";	//Set change bit
NETWORK
TITLE = Global End
      CLR;	//---Clear all commands
      =     #Ma.CmdOn;
      =     #Ma.CmdOff;
      =     #Ma.CmdNext;
      =     #Ma.CmdFaultReset;
      =     #Ma.CmdAirlockOff;
// 
//--- Interlocking pressure 
      A     #BlowOff.StLN;
      ON    #Ma.Par.ParWithBlowOff;
      AN    #AirlockA.StStartedFwd;
      AN    #AirlockB.StStartedFwd;
      A     #tmpBlowerStarted;
      =     #Pressure.InMonMinP;
      A     #Ma.InLocal;	//[5.7]
      AN    #Ma.InManual;	//[5.7]
      A     #tmpBlowerStopped;	//[5.7]
      =     #Pressure.InLocal;	//[5.7]
//--- InLocal high levels // [5.6] moved to Global End
      AN    #tmpWayA;
      A     #tmpWayB;
      O     #AirlockA.InLocal;
      =     #HLInletA.InLocal;
      AN    #tmpWayB;
      O     #AirlockB.InLocal;
      =     #HLInletB.InLocal;
//--- Interlocking HL        [6.2] moved to "global end"
      SET;
      S     #HLInletA.InMonFalse;
      S     #HLInletB.InMonFalse;
END_FUNCTION_BLOCK

FUNCTION_BLOCK "GCS7_M_PressureVessel"	// FB 68
TITLE = Pressure Vessel Conveying system
//  
//COPYRIGHT:    (C) 1999  BUEHLER AG, CH-9240 UZWIL, SWITZERLAND
//
//PRODUCT:      GCS7
//
//TITLE:        FB 68 Machine Control:Pressure Vessel Conveying System
//
//-------------------------------------------------------------------------
//
//IDENT:        AUTHOR:             DEPT:                       DATE:
//
//FB68.4.0      A. Egli             CT3                         17-Jun-2002
//              New Release with one block 
//FB68.3.2      A. Egli             CT3                         18-Apr-2000
//              Clearing time only if not InMinPrssure
//FB68.3.1      A. Egli             CT3                          2-Dec-1999
//              Conditon for RecycValve1 and RecycValve2
//FB68.3.0      A. Egli             CT3                         11-Oct-1999
//              Local data reduced
//FB68.2A       A. Egli             CT3                         04-Mai-1999
//              1st Release in S7
//
//-------------------------------------------------------------------------
//
//PURPOSE:      MANUAL : see [LL.TAKxxMAN]
//
//RESTRICTIONS: S7
//              ACCU2: Pointer to dynamic datas of the machine
//              ACCU1: Pointer to parameter datas of the machine
//
//-------------------------------------------------------------------------
//
AUTHOR : EA
FAMILY : GCS7LL
NAME : PulsePha
VERSION : 4.0
VAR
  Ma : UDT 20680;
  ConvValve1 : FB 13;	//Element
  FluidValve1 : FB 13;	//Element
  InletValve1 : FB 13;	//Element
  RecycValve1 : FB 13;	//Element
  OutletValve : FB 13;	//Element
  Vibro : FB 11;	//Element
  ConvValve2 : FB 13;	//Element
  FluidValve2 : FB 13;	//Element
  InletValve2 : FB 13;	//Element
  RecycValve2 : FB 13;	//Element
END_VAR
VAR_TEMP
  tmpEnable : BOOL ;
  tmpVKE : BOOL ;
  tmpEnableConveying : BOOL ;	//General condition for conveying Valve
  tmpAirOK : BOOL ;
  tmpLenDyn : INT ;
END_VAR
BEGIN
NETWORK
TITLE =
      L     42;
      T     #tmpLenDyn;
NETWORK
TITLE = PC Control
//=== Test Object number =====================
      L     "SYS_DirectCtrlDB".PC.ObjectNo;	//PCControl.ObjectNo
      L     #Ma.Par.ParObjectNo;	//Input ObjectNo
      <>I;
      JC    aEnd;
//=== Test OType      ========================
      L     2068;	//Input object type
      L     "SYS_DirectCtrlDB".PC.ObjectType;	//PCControl.ObjectType
      <>I;
      JC    aEnd;
//=== Test Handshake =========================
      A     "SYS_DirectCtrlDB".PC.Hsk.FExamine;	// Handshake.FExamine
      JC    aExa;
      A     "SYS_DirectCtrlDB".PC.Hsk.FDefineCmd;	// Handshake.FDefineCmd
      JC    aCmd;
      A     "SYS_DirectCtrlDB".PC.Hsk.FDefinePara;	// Handshake.FDefinePara
      JC    pPar;
aIni: L     2;	// FcInit
      UC    "SYS_DirectCtrl";
      JU    aEnd;
// Write parameter 
pPar: LAR1  P#DBX 58.0;
      L     P#6.0;
      +AR1;
      L     DBW [AR1,P#4.0];
      T     #Ma.Par.ParDelayFluidTime;
      L     DBW [AR1,P#6.0];
      T     #Ma.Par.ParMinConveyingTime;
      L     DBW [AR1,P#8.0];
      T     #Ma.Par.ParPulseBothTime;
      L     DBW [AR1,P#10.0];
      T     #Ma.Par.ParPulseFluidOnlyTime;
      L     DBW [AR1,P#12.0];
      T     #Ma.Par.ParClearingTime;
      L     DBW [AR1,P#14.0];
      T     #Ma.Par.ParPulseCnt;
// Write new commands from PC to Interface of group 
aCmd: A     "SYS_DirectCtrlDB".PC.Cmd1[8];	//CmdOff   
      S     #Ma.CmdOff;
      A     "SYS_DirectCtrlDB".PC.Cmd1[9];	//CmdConveying
      S     #Ma.CmdConveying;
      A     "SYS_DirectCtrlDB".PC.Cmd1[10];	//CmdNext
      S     #Ma.CmdNext;
      A     "SYS_DirectCtrlDB".PC.Cmd1[11];	//CmdFaultReset
      S     #Ma.CmdFaultReset;
      A     "SYS_DirectCtrlDB".PC.Cmd1[14];	//CmdFilling1
      S     #Ma.CmdFilling2;
      A     "SYS_DirectCtrlDB".PC.Cmd1[15];	//CmdFilling1
      S     #Ma.CmdFilling1;
      A     "SYS_DirectCtrlDB".PC.Cmd2[0];	//CmdPulsing
      S     #Ma.CmdPulsing;
      A     "SYS_DirectCtrlDB".PC.Cmd1[13];	//CmdManualOn
      S     #Ma.InManual;
      A     "SYS_DirectCtrlDB".PC.Cmd2[13];	//CmdManualOff
      R     #Ma.InManual;
      JU    aIni;
aExa: TAR2;	// Address Dynamic datas
      T     "SYS_DirectCtrlDB".GC.InDynAddr;	// -->PCControl.GC.InDynAddr
      L     #tmpLenDyn;	// Length Dynamic datas
      T     "SYS_DirectCtrlDB".GC.InDynLen;	// -->PCControl.GC.InDynLen
      L     0;
      T     "SYS_DirectCtrlDB".GC.InParaAddr;	// -->PCControl.GC.InParaAddr
      T     "SYS_DirectCtrlDB".GC.InParaLen;	// -->PCControl.GC.InParaLen
      L     1;	// Code FcExamine
      UC    "SYS_DirectCtrl";
      L     10;	//Revision
      T     "SYS_DirectCtrlDB".GC.Revision;
aEnd: NOP   0;
NETWORK
TITLE = Interlocking
//===Global Group Orders===
//===Global Group Orders===
      A     "GCS7_Gr_OutManualOn";	///Gr.OutManualOn
      S     #Ma.InManual;
      A     "GCS7_Gr_OutManualOff";	//Gr.OutManualOff
      R     #Ma.InManual;
      A     #Ma.InManual;
      S     "GCS7_Gr_InManual";	//Gr.InManual
//Fault 
      O     #ConvValve1.StFault;
      O     #FluidValve1.StFault;
      O     #InletValve1.StFault;
      O     #RecycValve1.StFault;
      O     #OutletValve.StFault;
      O     #Vibro.StFault;
      O     #ConvValve2.StFault;
      O     #FluidValve2.StFault;
      O     #InletValve2.StFault;
      O     #RecycValve2.StFault;
      =     #Ma.OutFault;
//Local
      A(;
      A     #OutletValve.StLN;
      ON    #Ma.Par.ParWithOutletValve;
      );
      A(;
      A     #RecycValve1.StLN;
      ON    #Ma.Par.ParWithRecycValve;
      );
      A     #InletValve1.StLN;
      A     #ConvValve1.StLN;
      A     #FluidValve1.StLN;
      A(;
      A     #RecycValve2.StLN;
      ON    #Ma.Par.ParWithRecycValve;
      A     #InletValve2.StLN;
      A     #ConvValve2.StLN;
      A     #FluidValve2.StLN;
      ON    #Ma.Par.ParType2Vessel;
      );
      A     #Ma.InLocal;
      AN    #Ma.InManual;
      S     #ConvValve1.InLocal;
      AN    #Ma.InLocal;
      O     #Ma.InManual;
      R     #ConvValve1.InLocal;
      A     #ConvValve1.InLocal;
      =     #FluidValve1.InLocal;
      =     #InletValve1.InLocal;
      =     #RecycValve1.InLocal;
      =     #OutletValve.InLocal;
      =     #Vibro.InLocal;
      =     #ConvValve2.InLocal;
      =     #FluidValve2.InLocal;
      =     #InletValve2.InLocal;
      =     #RecycValve2.InLocal;
//Enable 
      AN    #Ma.InLocal;
      O     #Ma.InManual;
      AN    #Ma.CmdOff;
      =     #tmpEnable;
//Temp flag
      A     #Ma.InAirOk;
      O     #Ma.InManual;
      =     #tmpAirOK;
//Manual filling
      A     #Ma.CmdFilling1;
      S     #Ma.Par.OutManFilling1;
      A     #Ma.CmdFilling2;
      S     #Ma.Par.OutManFilling2;
      AN    #Ma.InManual;
      O     #Ma.CmdOff;
      O     #Ma.CmdConveying;
      R     #Ma.Par.OutManFilling1;
      R     #Ma.Par.OutManFilling2;
NETWORK
TITLE = Call ConvValve1
      CALL  #ConvValve1;
NETWORK
TITLE = Call FluidValve1
      CALL  #FluidValve1;
NETWORK
TITLE = Call InletValve
      CALL  #InletValve1;
NETWORK
TITLE = Call OutletValve
      AN    #Ma.Par.ParWithOutletValve;
      JC    E05;
      CALL  #OutletValve;
NETWORK
TITLE = Call RecycValve
E05:  AN    #Ma.Par.ParWithRecycValve;
      JC    E06;
      CALL  #RecycValve1;
NETWORK
TITLE = Call Vibro
E06:  SET;
      S     #Vibro.Par.ParPulse;
// Call Vibro
      CALL  #Vibro;
NETWORK
TITLE = Call ConvValve2
      AN    #Ma.Par.ParType2Vessel;
      JC    StJ0;
      CALL  #ConvValve2;
NETWORK
TITLE = Call FluidValve2
      CALL  #FluidValve2;
NETWORK
TITLE = Call InletValve2
      CALL  #InletValve2;
NETWORK
TITLE = Call RecycValve2
      AN    #Ma.Par.ParWithRecycValve;
      JC    StJ0;
      CALL  #RecycValve2;
NETWORK
TITLE = Jump to actual state
StJ0: A     #Ma.StStopped;
      JC    S0;
      A     #Ma.StFilling;
      JC    S1;
      A     #Ma.StConveying;
      JC    S2;
      A     #Ma.StPulsing;
      JC    S3;
      A     #Ma.StClearing;
      JC    S5;
      A     #Ma.StCleared;
      JC    S6;
      JU    xxS6;	// ===> Initialisation
NETWORK
TITLE = Stopped
//any Transition 
xxS0: S     #Ma.StStopped;
      JU    OUT;
//=== Logic
S0:   A(;
      A     #Ma.InEnableFilling1;
      AN    #Ma.InManual;
      O;
      A     #Ma.InEnableFilling2;
      AN    #Ma.InManual;
      );
      A     #Ma.CmdNext;
      O     #Ma.CmdFilling1;
      O     #Ma.CmdFilling2;
      R     #Ma.StStopped;
      JC    xxS1;	//-->StFilling
      A     #Ma.InEnableConveying;
      AN    #Ma.InManual;
      A     #Ma.CmdNext;
      O     #Ma.CmdConveying;
      R     #Ma.StStopped;
      JC    xxS2;	//-->Conveying
      JU    OUT;
NETWORK
TITLE = StFilling
//any Transition 
xxS1: S     #Ma.StFilling;
      S     #Ma.OutLoaded;
//=== Logic
S1:   AN    #Ma.InEnableFilling1;
      AN    #Ma.InEnableFilling2;
      AN    #Ma.InManual;
      O     #Ma.CmdOff;
      R     #Ma.StFilling;
      JC    xxS0;	//--> StStopped
      A     #Ma.CmdConveying;
      R     #Ma.StFilling;
      JC    xxS2;	//--> StConveying
      JU    OUT;
NETWORK
TITLE = StConveying
//any Transition 
xxS2: S     #Ma.StConveying;
      R     #Ma.Par.OutDelayFluidDone;
      R     #Ma.Par.OutConvTimeDone;
      L     0;
      T     #Ma.Par.OutDelayFluidTime;
      T     #Ma.Par.OutConveyingTime;
//=== Logic
// Condition for Stopped
S2:   A     #Ma.InNoRestdischarge;
      A     #Ma.Par.OutConvTimeDone;
      AN    #Ma.InMaxPressure;
      AN    #Ma.InMinPressure;
      AN    #Ma.InManual;
      R     #Ma.StConveying;
      JC    xxS6;	//--> StCleared;
      ON    #Ma.InEnableConveying;
      AN    #Ma.InManual;
      O     #Ma.CmdOff;
      R     #Ma.StConveying;
      JC    xxS0;	//--> StStopped
// Condition for Fluidization
      A     #Ma.Par.OutConvTimeDone;
      AN    #Ma.InMaxPressure;
      AN    #Ma.InMinPressure;
      AN    #Ma.InManual;
      O;
      A     #Ma.CmdPulsing;
      R     #Ma.StConveying;
      JC    xxS3;	//--> StPulsing
// Condition for Filling
      A     #Ma.CmdFilling1;
      O     #Ma.CmdFilling2;
      R     #Ma.StConveying;
      JC    xxS1;	//--> StFilling
//Delay time fluidization valve
      A     #OutletValve.StHN;
      ON    #Ma.Par.ParWithOutletValve;
      A     #ConvValve1.StHN;
      A(;
      A     #ConvValve2.StHN;
      ON    #Ma.Par.ParType2Vessel;
      );
      A     #tmpAirOK;
      AN    #Ma.OutBlowoff;
      JC    S2FL;
      R     #Ma.Par.OutDelayFluidDone;
      R     #Ma.Par.OutConvTimeDone;
      L     0;
      T     #Ma.Par.OutDelayFluidTime;
      T     #Ma.Par.OutConveyingTime;
      JU    OUT;
S2FL: A     #Ma.Par.OutDelayFluidDone;
      JC    S2B1;
      AN    "GCS7_Gr_OutTick200ms";	//Gr.OutTick200ms
      JC    S2A2;
      L     #Ma.Par.OutDelayFluidTime;
      +     2;
      T     #Ma.Par.OutDelayFluidTime;
S2A2: L     #Ma.Par.ParDelayFluidTime;
      L     #Ma.Par.OutDelayFluidTime;
      <=I;
      S     #Ma.Par.OutDelayFluidDone;
//Conveying time
S2B1: A     #Ma.Par.OutConvTimeDone;
      JC    S2H2;
      A     #OutletValve.StHN;
      ON    #Ma.Par.ParWithOutletValve;
      A(;
      A     #RecycValve1.StLN;
      ON    #Ma.Par.ParWithRecycValve;
      );
      A     #InletValve1.StLN;
      A     #ConvValve1.StHN;
      A     #FluidValve1.StHN;
      A(;
      A     #RecycValve2.StLN;
      ON    #Ma.Par.ParWithRecycValve;
      A     #InletValve2.StLN;
      A     #ConvValve2.StHN;
      A     #FluidValve2.StHN;
      ON    #Ma.Par.ParType2Vessel;
      );
      A     #tmpAirOK;
      AN    #Ma.OutBlowoff;
      JCN   OUT;
      AN    "GCS7_Gr_OutTick200ms";	//Gr.OutTick200ms
      JC    S3B2;
      L     #Ma.Par.OutConveyingTime;
      +     2;
      T     #Ma.Par.OutConveyingTime;
      L     #Ma.Par.ParMinConveyingTime;
      L     #Ma.Par.OutConveyingTime;
      <=I;
      S     #Ma.Par.OutConvTimeDone;
S2H2: JU    OUT;
NETWORK
TITLE = StPulsing
//any Transition 
xxS3: S     #Ma.StPulsing;
      S     #Ma.Par.OutPulseFluidOnly;
      L     0;
      T     #Ma.Par.OutPulseCnt;
      T     #Ma.Par.OutPulseTime;
//=== Logic
// Condition for Clearing
S3:   L     #Ma.Par.ParPulseCnt;
      L     #Ma.Par.OutPulseCnt;
      <=I;
      AN    #Ma.InManual;
      R     #Ma.StPulsing;
      JC    xxS5;	//--> StClearing
// Condition for Conveying
      A     #Ma.CmdConveying;
      R     #Ma.Par.OutPulseFluidOnly;
      R     #Ma.StPulsing;
      JC    xxS2;	//--> StConveying
// Condition for Stopped
      AN    #Ma.InEnableConveying;
      AN    #Ma.InManual;
      O     #Ma.CmdOff;
      R     #Ma.Par.OutPulseFluidOnly;
      R     #Ma.StPulsing;
      JC    xxS0;	//--> StStopped
// Condition for Filling
      A     #Ma.CmdFilling1;
      O     #Ma.CmdFilling2;
      R     #Ma.StPulsing;
      R     #Ma.Par.OutPulseFluidOnly;
      JC    xxS1;	//--> StFilling
//PulseBothTime
      A     #OutletValve.StHN;
      ON    #Ma.Par.ParWithOutletValve;
      A(;
      A     #RecycValve1.StLN;
      ON    #Ma.Par.ParWithRecycValve;
      );
      A     #FluidValve1.StHN;
      A     #InletValve1.StLN;
      A(;
      A     #RecycValve2.StLN;
      ON    #Ma.Par.ParWithRecycValve;
      A     #FluidValve2.StHN;
      A     #InletValve2.StLN;
      ON    #Ma.Par.ParType2Vessel;
      );
      A     #tmpAirOK;
      AN    #Ma.OutBlowoff;
      NOT;
      R     #Ma.Par.OutPulseFluidOnly;
      JC    OUT;
      A     #Ma.Par.OutPulseFluidOnly;
      JC    S3B1;
      AN    "GCS7_Gr_OutTick200ms";	//Gr.OutTick200ms
      JC    S3A2;
      L     #Ma.Par.OutPulseTime;
      +     2;
      T     #Ma.Par.OutPulseTime;
S3A2: L     #Ma.Par.ParPulseBothTime;
      L     #Ma.Par.OutPulseTime;
      >I;
      JC    OUT;
      S     #Ma.Par.OutPulseFluidOnly;
      L     0;
      T     #Ma.Par.OutPulseTime;
      L     #Ma.Par.OutPulseCnt;
      +     1;
      T     #Ma.Par.OutPulseCnt;
      JU    OUT;
//PulseFluidOnlyTime
S3B1: AN    "GCS7_Gr_OutTick200ms";	//Gr.OutTick200ms
      JC    S3B2;
      L     #Ma.Par.OutPulseTime;
      +     2;
      T     #Ma.Par.OutPulseTime;
S3B2: L     #Ma.Par.ParPulseFluidOnlyTime;
      L     #Ma.Par.OutPulseTime;
      >I;
      JC    OUT;
      R     #Ma.Par.OutPulseFluidOnly;
      S     #Vibro.CmdNext;
      L     0;
      T     #Ma.Par.OutPulseTime;
      JU    OUT;
NETWORK
TITLE = StClearing
//any Transition 
xxS5: S     #Ma.StClearing;
      L     0;
      T     #Ma.Par.OutClearingTime;
//=== Logic
// Condition for StCleared
S5:   L     #Ma.Par.ParClearingTime;
      L     #Ma.Par.OutClearingTime;
      <=I;
      R     #Ma.StClearing;
      JC    xxS6;	//--> StCleared;
// Condition for StConveying
      A     #Ma.InManual;
      R     #Ma.StClearing;
      JC    xxS2;	//--> StConveying
// Condition for StStopped
      AN    #Ma.InEnableConveying;
      R     #Ma.StClearing;
      JC    xxS0;	//--> StStopped
//Clearing Time
      AN    "GCS7_Gr_OutTick200ms";	//Gr.OutTick200ms
      O     #Ma.InMinPressure;	//[3.2]
      O     #Ma.OutFault;
      JC    OUT;
      L     #Ma.Par.OutClearingTime;
      +     2;
      T     #Ma.Par.OutClearingTime;
      JU    OUT;
NETWORK
TITLE = StCleared
//any Transition 
xxS6: S     #Ma.StCleared;
      R     #Ma.OutLoaded;
      JU    OUT;
//=== Logic
//Condition for StFilling
S6:   A     #Ma.InEnableFilling1;
      O     #Ma.InEnableFilling2;
      R     #Ma.StCleared;
      JC    xxS1;	//-->StFilling
//Condition for StConveying
      A     #Ma.CmdConveying;
      R     #Ma.StCleared;
      JC    xxS2;	//-->StConveying
// Condition for StStopped
      AN    #Ma.InEnableConveying;
      O     #Ma.InManual;
      R     #Ma.StCleared;
      JC    xxS0;	//--> StStopped
      JU    OUT;
NETWORK
TITLE = State Code
// State           StCode
// ----------------------
// StFault            32
// StStopped          1
// StFilling          2
// StConveying        3
// StPulsing          4
// StClearing         5
// StCleared          6
OUT:  A     #Ma.OutFault;
      L     32;	//Code=Fault
      JC    Code;
      A     #Ma.StStopped;
      L     1;	//Code=Stopped
      JC    Code;
      L     2;	//Code=Filling
      A     #Ma.StFilling;
      JC    Code;
      L     3;	//Code=Conveying
      A     #Ma.StConveying;
      JC    Code;
      L     4;	//Code=Pulsing
      A     #Ma.StPulsing;
      JC    Code;
      L     5;	//Code=Clearing
      A     #Ma.StClearing;
      JC    Code;
      L     6;	//Code=Cleared
Code: L     #Ma.StCode;	// Old state code
      TAK;
      T     #Ma.StCode;	// Save state code
      <>I;
      L     3;
      UC    "SYS_CBitCtrl";	//Set change bit
NETWORK
TITLE = General
      A     #Ma.CmdFaultReset;
      S     #ConvValve1.CmdFaultReset;
      S     #FluidValve1.CmdFaultReset;
      S     #InletValve1.CmdFaultReset;
      S     #OutletValve.CmdFaultReset;
      S     #RecycValve1.CmdFaultReset;
      S     #Vibro.CmdFaultReset;
      S     #ConvValve2.CmdFaultReset;
      S     #FluidValve2.CmdFaultReset;
      S     #InletValve2.CmdFaultReset;
      S     #RecycValve2.CmdFaultReset;
//RecycValve 
      A     #Ma.InEnableFilling1;
      AN    #Ma.InManual;
      O     #Ma.Par.OutManFilling1;
      A(;	//[3.1] 
      A     #OutletValve.StLN;
      ON    #Ma.Par.ParWithOutletValve;
      );	//[3.1]
      A     #FluidValve1.StLN;
      A     #ConvValve1.StLN;
      A     #Ma.StFilling;
      =     #RecycValve1.InEnableHN;
      R     #RecycValve1.InEnableLN;
      AN    #RecycValve1.InEnableHN;
      =     #RecycValve1.InEnableLN;
//RecycValve2 
      A     #Ma.InEnableFilling2;
      AN    #Ma.InManual;
      O     #Ma.Par.OutManFilling2;
      A(;	//[3.1]
      A     #OutletValve.StLN;
      ON    #Ma.Par.ParWithOutletValve;
      );	//[3.1]
      A     #FluidValve2.StLN;
      A     #ConvValve2.StLN;
      A     #Ma.StFilling;
      =     #RecycValve2.InEnableHN;
      R     #RecycValve2.InEnableLN;
      AN    #RecycValve2.InEnableHN;
      =     #RecycValve2.InEnableLN;
//Inlet Valve 
      A     #RecycValve1.StHN;
      ON    #Ma.Par.ParWithRecycValve;
      A     #RecycValve1.InEnableHN;
      =     #InletValve1.InEnableHN;
      AN    #InletValve1.InEnableHN;
      =     #InletValve1.InEnableLN;
//InletValve2
      A     #RecycValve2.StHN;
      ON    #Ma.Par.ParWithRecycValve;
      A     #RecycValve2.InEnableHN;
      =     #InletValve2.InEnableHN;
      AN    #InletValve2.InEnableHN;
      =     #InletValve2.InEnableLN;
//Outlet Valve 
      A     #Ma.InEnableConveying;
      O     #Ma.InManual;
      AN    #Ma.StStopped;
      AN    #Ma.StFilling;
      AN    #Ma.StCleared;
      =     #OutletValve.InEnableHN;
      R     #OutletValve.InEnableLN;
      AN    #OutletValve.InEnableHN;
      A     #FluidValve1.StLN;
      A     #ConvValve1.StLN;
      S     #OutletValve.InEnableLN;
//Conveying valve and fluidization valve
      A     #Ma.StConveying;
      O     #Ma.StPulsing;
      O     #Ma.StClearing;
      AN    #Ma.OutFault;
      A(;
      A     #OutletValve.StHN;
      ON    #Ma.Par.ParWithOutletValve;
      );
      A(;
      A     #RecycValve1.StLN;
      ON    #Ma.Par.ParWithOutletValve;
      );
      A     #InletValve1.StLN;
      A(;
      A     #RecycValve2.StLN;
      ON    #Ma.Par.ParWithOutletValve;
      A     #InletValve2.StLN;
      ON    #Ma.Par.ParType2Vessel;
      );
      A(;
      A     #Ma.InEnableConveying;
      O     #Ma.InManual;
      );
      AN    #Ma.InOverPressure;
      =     #tmpEnableConveying;
//FluidValve / FluidValve2
      AN    #Ma.StConveying;
      O     #Ma.Par.OutDelayFluidDone;
      AN    #Ma.InMaxPressure;
      A     #tmpEnableConveying;
      =     #FluidValve1.InEnableHN;
      AN    #tmpEnableConveying;
      O     #Ma.InMaxPressure;
      =     #FluidValve1.InEnableLN;
      A     #FluidValve1.InEnableHN;
      =     #FluidValve2.InEnableHN;
      A     #FluidValve1.InEnableLN;
      =     #FluidValve2.InEnableLN;
//ConvValve / ConvValve2 
      AN    #Ma.Par.OutPulseFluidOnly;
      ON    #Ma.StPulsing;
      A     #tmpEnableConveying;
      =     #ConvValve1.InEnableHN;
      AN    #ConvValve1.InEnableHN;
      A(;
      A     #Ma.InBlowoffIsOpen;
      O     #Ma.StPulsing;
      );
      =     #ConvValve1.InEnableLN;
      A     #ConvValve1.InEnableHN;
      =     #ConvValve2.InEnableHN;
      A     #ConvValve1.InEnableLN;
      =     #ConvValve2.InEnableLN;
//Vibro
      SET;
      =     #Vibro.InEnable;
//Blow off 
      AN    #Ma.StConveying;
      AN    #Ma.StPulsing;
      AN    #Ma.StClearing;
      O     #Ma.InOverPressure;
      O     #Ma.OutFault;
      O;
      A     #FluidValve1.StLN;
      AN    #ConvValve1.StHN;
      =     #Ma.OutBlowoff;
//OutEnableFilling
//        U       RecycValve1.InEnableHN;
//        U(;
//        U       RecycValve1.StHN;
//        ON      #Ma.Par.ParWithRecycValve;
//        );
//        U       InletValve1.StHN;
//        =       Ma.OutEnableFilling;
//OutEnableBlower
      A     #OutletValve.StHN;
      ON    #Ma.Par.ParWithOutletValve;
      A(;
      A     #FluidValve1.StHN;
      O     #ConvValve1.StHN;
      );
      AN    #ConvValve1.StFault;
      A(;
      A     #FluidValve2.StHN;
      O     #ConvValve2.StHN;
      AN    #ConvValve2.StFault;
      ON    #Ma.Par.ParType2Vessel;
      );
      O     #Ma.InBlowoffIsOpen;
      =     #Ma.OutEnableBlower;
NETWORK
TITLE = Global End
//Next
      SET;
      S     #ConvValve1.CmdNext;
      S     #FluidValve1.CmdNext;
      S     #OutletValve.CmdNext;
      S     #InletValve1.CmdNext;
      S     #RecycValve1.CmdNext;
      S     #ConvValve2.CmdNext;
      S     #FluidValve2.CmdNext;
      S     #InletValve2.CmdNext;
      S     #RecycValve2.CmdNext;
//---Clear all commands
      CLR;
      =     #Ma.CmdOff;
      =     #Ma.CmdNext;
      =     #Ma.CmdFaultReset;
      =     #Ma.CmdConveying;
      =     #Ma.CmdPulsing;
      =     #Ma.CmdFilling1;
      =     #Ma.CmdFilling2;
// 
END_FUNCTION_BLOCK

FUNCTION_BLOCK "GCS7_M_RotaryDis"	// FB 69
TITLE = Rotary
//  
//COPYRIGHT:    (C) 1997  BUHLER AG, CH-9240 UZWIL,  SWITZERLAND
//
//PRODUCT:      GCS7
//
//TITLE:        FB 69 MACHINE-CONTROL: Rotary
//
//-------------------------------------------------------------------------
//
//IDENT:        AUTHOR:             DEPT:                       DATE:
//FB69.4.2      A. Egli             CT3                         14-Sep-2006
//              Set OutRev
//FB69.4.1      A. Egli             CT3                         12-Sep-2003
//              Reset Ma.OutFlagAdjusted in state StFault
//FB69.4.0      A. Egli             CT3                         17-Jun-2002
//              New Release with one block 
//FB69.3.0      A.Egli              CT3                         11-Oct-1999
//              New ident type
//FB69.2B       K. Tischer          MU664                       06-Mrz-1999
//              CC FC2 not UC FC2
//FB69.2A       A. Egli             CT3                         04-Mai-1998
//              StFault = StCode 32
//FB69.1A       A.Egli              AEE61                       05-Jul-1997
//              1st Release in S7
//
//-------------------------------------------------------------------------
//
//PURPOSE:      MANUAL : see [LL.ROTxxMAN]
//
//RESTRICTIONS: S7
//              ACCU2: Pointer to dynamic datas of the machine
//              ACCU1: Pointer to parameter datas of the machine
//
//-------------------------------------------------------------------------
//
AUTHOR : EA
FAMILY : GCS7LL
NAME : Rotary
VERSION : 4.2
VAR
  Ma : UDT 20690;
  Motor : FB 12;	//Element
  Mon : FB 14;	//Element
END_VAR
VAR_TEMP
  tmpFaultStop : BOOL ;
  tmpFaultSum : BOOL ;
  tmpLocal : BOOL ;
  tmpEnable : BOOL ;
  tmpInPosition : BOOL ;
  tmpPosition : BOOL ;
  tmpCnt : INT ;
  tmpAnyPosition : BOOL ;
  tmp2LS : BOOL ;	// 2 or more LS pressed
  tmpFlagNewPosition : BOOL ;
  tmpPrevPos : BOOL ;	// Actual position is before target position
  tmpSetPos : DWORD ;
  tmpLastPos : DWORD ;
  tmpLenDyn : INT ;
END_VAR
BEGIN
NETWORK
TITLE =
      L     32;
      T     #tmpLenDyn;
NETWORK
TITLE = PC Control
//=== Test Object number =====================
      L     "SYS_DirectCtrlDB".PC.ObjectNo;	//PCControl.ObjectNo
      L     #Ma.Par.ParObjectNo;	//Input ObjectNo
      <>I;
      JC    aEnd;
//=== Test OType      ========================
      L     2069;	//Input object type
      L     "SYS_DirectCtrlDB".PC.ObjectType;	//PCControl.ObjectType
      <>I;
      JC    aEnd;
//=== Test Handshake =========================
      A     "SYS_DirectCtrlDB".PC.Hsk.FExamine;	// Handshake.FExamine
      JC    aExa;
      A     "SYS_DirectCtrlDB".PC.Hsk.FDefineCmd;	// Handshake.FDefineCmd
      O     "SYS_DirectCtrlDB".PC.Hsk.FDefinePara;	// Handshake.FDefinePara
      JC    aCmd;
aIni: L     2;	// FcInit
      UC    "SYS_DirectCtrl";
      JU    aEnd;
// Write new commands from PC to Interface of group 
aCmd: A     "SYS_DirectCtrlDB".PC.Cmd1[8];	//Cmd1[8]=CmdOff
      S     #Ma.CmdOff;
      A     "SYS_DirectCtrlDB".PC.Cmd1[9];	//Cmd1[9]=CmdOn
      S     #Ma.CmdOn;
      A     "SYS_DirectCtrlDB".PC.Cmd1[10];	//Cmd1[10]=CmdNext
      S     #Ma.CmdNext;
      A     "SYS_DirectCtrlDB".PC.Cmd1[11];	//Cmd1[11]=CmdFaultReset
      S     #Ma.CmdFaultReset;
      A     "SYS_DirectCtrlDB".PC.Cmd1[13];	//Cmd1[13]=CmdManualOn
      S     #Ma.InManual;
      A     "SYS_DirectCtrlDB".PC.Cmd2[13];	//Cmd2[13]=CmdManualOff
      R     #Ma.InManual;
      A     "SYS_DirectCtrlDB".PC.Cmd1[14];	//Cmd1[14]=CmdPrevPos
      S     #Ma.CmdPrevPos;
      A     "SYS_DirectCtrlDB".PC.Cmd1[15];	//Cmd1[15]=CmdNextPos
      S     #Ma.CmdNextPos;
      AN    "SYS_DirectCtrlDB".PC.Hsk.FDefinePara;	// Handshake.FDefinePara
      JC    aIni;
      JU    aIni;
aExa: TAR2;	// Address Dynamic datas
      T     "SYS_DirectCtrlDB".GC.InDynAddr;	// -->PCControl.GC.InDynAddr
      L     #tmpLenDyn;	// Length Dynamic datas
      T     "SYS_DirectCtrlDB".GC.InDynLen;	// -->PCControl.GC.InDynLen
      L     0;
      T     "SYS_DirectCtrlDB".GC.InParaAddr;	// -->PCControl.GC.InParaAddr
      T     "SYS_DirectCtrlDB".GC.InParaLen;	// -->PCControl.GC.InParaLen
      L     1;	// Code FcExamine
      UC    "SYS_DirectCtrl";
      L     10;	//Revision
      T     "SYS_DirectCtrlDB".GC.Revision;
aEnd: NOP   0;
NETWORK
TITLE = Interlocking 1 
//===Global Group Orders===
      A     "GCS7_Gr_OutManualOn";	//Gr.OutManualOn
      S     #Ma.InManual;
      A     "GCS7_Gr_OutManualOff";	//Gr.OutManualOff
      R     #Ma.InManual;
      A     #Ma.InManual;
      S     "GCS7_Gr_InManual";	//Gr.InManual
//----
      A     #Ma.InLocal;
      AN    #Ma.InManual;
      =     #tmpLocal;
NETWORK
TITLE = Set position
      L     #Ma.OutSetPos;	// Ma.OutSetPos[1..32] 
      T     #tmpSetPos;
      L     #Ma.Par.ParNoOfPosition;
      L     1;
      RLD;	//Last position
      RRD   1;
      T     #tmpLastPos;
      A     #Ma.InManual;
      JC    INJ1;
//    Automatic
      L     #Ma.InSetPos;	// Ma.InpSetPos[1..32] 
      JU    INJx;	//-->Set position
//    Manual
INJ1: AN    #Ma.CmdPrevPos;
      JC    INJ3;
      S     #Ma.OutFlagChange;
      L     1;	// Fist position  
      L     #Ma.OutSetPos;	// Ma.OutSetPos[1..32] 
      CAD;
      ==D;
      L     #tmpLastPos;
      JC    INJe;	//-->  goto last position
      TAK;
      RRD   1;
      CAD;
      JU    INJx;
INJ3: AN    #Ma.CmdNextPos;
      JC    IN2;
      S     #Ma.OutFlagChange;
      L     #tmpLastPos;
      CAD;
      L     #Ma.OutSetPos;	// Ma.OutSetPos[1..32] 
      ==D;
      L     1;	//--> goto first pos
      JC    INJe;
      L     #Ma.OutSetPos;	// Ma.OutSetPos[1..32] 
      CAD;
      RLD   1;
INJe: CAD;
INJx: T     #Ma.OutSetPos;	// Ma.OutSetPos[1..32] 
//--- Test ---
IN2:  L     0;
      L     #Ma.OutSetPos;	// Ma.OutSetPos[1..32] 
      ==D;
      L     1;	//--> First position
      CAD;
      JC    INJx;
      L     32;
      L     #Ma.Par.ParNoOfPosition;
      ==I;
      JC    IN3;
      L     #tmpLastPos;
      L     #Ma.OutSetPos;	// Ma.OutSetPos[1..32] 
      CAD;
      <D;
      TAK;
      CAD;
      JC    INJx;	//--> Set last position
//---Test modification set position
IN3:  L     #Ma.OutSetPos;	// Ma.OutSetPos[1..32] 
      L     #tmpSetPos;
      <>D;
      =     #tmpFlagNewPosition;
//---Test actual position 
      LAR1  AR2;
      SET;
      R     #tmpAnyPosition;
      R     #tmp2LS;
      L     32;
LOP:  T     #tmpCnt;
      A     DIX [AR1,P#10.0];	// Ma.InpLSPos[1..32] 
      A     #tmpAnyPosition;
      S     #tmp2LS;	//--> Fault 2 LS
      AN    DIX [AR1,P#14.0];	// Ma.OutSetPos[1..32] 
      JC    L2;
L2:   A     DIX [AR1,P#10.0];	// Ma.InpLSPos[1..32] 
      S     #tmpAnyPosition;
      +AR1  P#0.1;
      L     #tmpCnt;
      LOOP  LOP;
      A     #tmp2LS;
      R     #tmpAnyPosition;
      L     #Ma.OutSetPos;	// Ma.OutSetPos[1..32] 
      CAD;
      L     #Ma.InpLSPos;	// Ma.InpLSPos[1..32] 
      CAD;
      ==D;
      A     #tmpAnyPosition;
      =     #tmpInPosition;
      >D;
      A     #tmpAnyPosition;
      =     #tmpPrevPos;
      A     #tmpLocal;	//[4.2]
      AN    #tmpInPosition;	//[4.2]
      O     #tmpFlagNewPosition;	//[4.2]
      R     #Ma.OutFlagAdjusted;	//[4.2]
      S     #Ma.OutRev;	//[4.2]--> Reverse     
NETWORK
TITLE = Interlocking 2
//--- Fault----
      A     #Mon.StFault;
      O     #Motor.StFault;
      =     #tmpFaultSum;
      =     #tmpFaultStop;
//--- Local mode --
      A     #tmpLocal;
      =     #Motor.InLocal;
      =     #Mon.InLocal;
//--- Fault Reset -------------
      A     #Ma.CmdFaultReset;
      S     #Motor.CmdFaultReset;
      S     #Mon.CmdFaultReset;
//--- Motor ---------
      A     #tmpPrevPos;
      A     #tmpAnyPosition;
      O     #Ma.InpLSPos[1];
      ON    #Ma.Par.Par2Dir;
      R     #Ma.OutRev;	//--> Reverse
      A     #Motor.OutpRunRev;
      S     #Ma.OutFlagChange;
      A     #tmpInPosition;
      AN    #Ma.OutRev;
      S     #Ma.OutFlagAdjusted;
      A     #Ma.InEnable;
      AN    #Ma.OutFlagAdjusted;
      O     #Ma.InManual;
      AN    #Ma.StFault;
      AN    #Ma.CmdOff;
      =     #tmpEnable;
// Forward
      AN    #Ma.OutRev;
      AN    #tmpInPosition;
      A     #tmpEnable;
      =     #Motor.InEnableFwd;
// Reverse
      A     #tmpEnable;
      A     #Ma.OutRev;
      A     #Ma.Par.Par2Dir;
      =     #Motor.InEnableRev;
// Next
      A     #Ma.CmdNext;
      AN    #Ma.InManual;
      O;
      A     #Ma.InManual;
      A     #Ma.CmdPrevPos;
      O;
      A     #Ma.InManual;
      A     #Ma.CmdNextPos;
      O     #Ma.CmdOn;
      O     #Ma.OutFlagChange;
      S     #Motor.CmdNext;
      AN    #tmpEnable;
      O     #Motor.OutpRunFwd;
      R     #Ma.OutFlagChange;
//--- Mon -----------
      A     #Motor.StStartedFwd;
      O     #Motor.StStartedRev;
      O     #Ma.OutFlagAdjusted;
      AN    #tmpFlagNewPosition;
      AN    #Ma.CmdFaultReset;	//***
      =     #Mon.InMonTrue;
      CLR;
      =     #Mon.InMonFalse;
// 
      A     #tmpInPosition;
      =     #Mon.InpTrue;
NETWORK
TITLE = Call Motor
      CALL  #Motor;
NETWORK
TITLE = Call Digital Input: Monitor B1
//Modify element parameter
      AN    #Ma.OutFlagAdjusted;
      AN    #tmpFlagNewPosition;
      =     #Mon.Par.Par2WorkingCond;
      SET;
      S     #Mon.Par.ParFaultRetry;
// Call element
      CALL  #Mon;
NETWORK
TITLE = Jump to actual state
      A     #Ma.StStopped;
      JC    S0;	// ===> State
      A     #Ma.StAdjusted;
      JC    S2;	// ===> State
      A     #Ma.StAdjusting;
      JC    S1;	// ===> State
      A     #Ma.StNoPosition;
      JC    S3;	// ===> State
      A     #Ma.StFault;
      JC    S4;	// ===> State
NETWORK
TITLE = Stopped
xxS0: S     #Ma.StStopped;
S0:   A     #tmpFaultSum;
      R     #Ma.StStopped;
      JC    xxS4;	//--> StFault
      AN    #Motor.StStopped;
      R     #Ma.StStopped;
      JC    xxS1;	//--> StAdjusting
// Condition for StAdjusted
      A     #tmpInPosition;
      R     #Ma.StStopped;
      JC    xxS2;	//--> StAdjusted
// Condition for StNoPosition
      AN    #tmpAnyPosition;
      R     #Ma.StStopped;
      JC    xxS3;	//--> StNoPosition
      JU    OUT;
NETWORK
TITLE = StAdjusting
xxS1: S     #Ma.StAdjusting;
S1:   A     #tmpFaultSum;
      R     #Ma.StAdjusting;
      JC    xxS4;	//--> StFault
// Condition for StAdjusted
      A     #tmpInPosition;
      AN    #Ma.OutRev;
      R     #Ma.StAdjusting;
      JC    xxS2;	//--> StAdjusted
// Condition for StNoPosition
      A     #Motor.StStopped;
      R     #Ma.StAdjusting;
      JC    xxS3;	//--> StNoPosition
      JU    OUT;
NETWORK
TITLE = StAdjusted
xxS2: S     #Ma.StAdjusted;
      S     #Ma.OutFlagAdjusted;
S2:   A     #tmpFaultSum;
      R     #Ma.StAdjusted;
      JC    xxS4;	//--> StFault
// Condition for StNoPosition
      AN    #tmpAnyPosition;
      R     #Ma.StAdjusted;
      JC    xxS3;	//--> StNoPosition
// Condition for StStopped
      AN    #tmpInPosition;
      R     #Ma.StAdjusted;
      JC    xxS3;	//--> StStopped
      JU    OUT;
NETWORK
TITLE = StNoPosition
xxS3: S     #Ma.StNoPosition;
S3:   A     #tmpFaultSum;
      R     #Ma.StNoPosition;
      JC    xxS4;	//--> StFault
// Condition for StStopped
      A     #tmpAnyPosition;
      R     #Ma.StNoPosition;
      JC    xxS0;	//--> StStopped
// Condition for StAdjusting
      AN    #Motor.StStopped;
      R     #Ma.StNoPosition;
      JC    xxS1;	//--> StAdjusting
      JU    OUT;
NETWORK
TITLE = Fault
xxS4: S     #Ma.StFault;
      R     #Ma.OutFlagAdjusted;
      S     #Ma.OutRev;	//--> Reverse
S4:   AN    #tmpFaultSum;
      R     #Ma.OutFlagAdjusted;	//[4.1]
      R     #Ma.StFault;
      JC    xxS3;	//--> StNoPosition
      JU    OUT;
OUT:  NOP   0;
NETWORK
TITLE = Global End
      CLR;	//---Clear all commands
      =     #Ma.CmdOff;
      =     #Ma.CmdOn;
      =     #Ma.CmdNext;
      =     #Ma.CmdFaultReset;
      =     #Ma.CmdPrevPos;
      =     #Ma.CmdNextPos;
NETWORK
TITLE = State Code
//Started
      L     3;	// StCode=Adjsuted
      A     #Ma.StAdjusted;
      JC    Code;
      L     1;	// StCode=Stopped
      A     #Ma.StStopped;
      JC    Code;
      L     2;	// StCode=Adjusting
      A     #Ma.StAdjusting;
      JC    Code;
      L     5;	// StCode=StNoPosition
      A     #Ma.StNoPosition;
      JC    Code;
      L     32;	// StCode=Fault
Code: L     #Ma.StCode;	// Old state code
      TAK;
      T     #Ma.StCode;	// Save state code
      <>I;
      L     3;
      CC    "SYS_CBitCtrl";	//Set change bit
END_FUNCTION_BLOCK

FUNCTION_BLOCK "GCS7_AddWayPattern"	// FB 70
TITLE = Add way pattern
//  
//COPYRIGHT:    (C) 1998  BUHLER AG , CH-9240 UZWIL  SWITZERLAND
//
//PRODUCT:      GCS7
//
//TITLE:        FB 90 Add Way Pattern 
//              (GCPROVB Revision 4)
//-------------------------------------------------------------------------
//
//IDENT:        AUTHOR:             DEPT:                       DATE:
//FB70.4.4      A.Egli              CT3                        30-Oct-2007
//              Start AdjustTime also at end of the AddTime
//FB70.4.3      A.Egli              CT3                        04-Oct-2007
//              BKT: Flap below slide are changing immediatly
//FB70.4.2      A.Egli              CT3                        23-Feb-2005
//              OutNewWayIsLonger only when InBKT
//FB70.4.1      A.Egli              CT3                        20-Jan-2005
//              Reset OutOldWayOK as long old pattern is 0 (reload software)
//FB70.4.0      A.Egli              CT3                        19-Nov-2004
//              InBKT : Close slide gate in shorter way as soon
//                      new way is open 
//FB70.3.1      A.Egli              CT3                         1-Apr-2002
//              Deselect old flaps
//FB70.3.0      A.Egli              CT3                        23-Okt-2002
//              Redesign
//FB70.2.2      Ph. Engler          MU664                      28-Dec-2000
//              Type Asp-Flaps (No ParBlowline) corrected
//              In case of a new receiver change during the
//              old and new pattern was active the new flap
//              has been closed.
//FB70.2.1      A.Egli              CT3                        17-Mai-2000
//              ParBlowLine
//FB70.2A       E.Hanselmann        AEMU664                    01-Feb-2000
//              Sequenz adjusting
//FB70.1A       A.Egli              CT3                        22-Jan-1998
//              1st Release in S7
//
//-------------------------------------------------------------------------
//
//PURPOSE:      MANUAL : see [LL.WAYxxMAN]
//
//RESTRICTIONS: S7
//-------------------------------------------------------------------------
//
//
//Input:
// 
//   InPointerPattern : Must pointer to Struct
//
//   Way : STRUCT 
//    InAdjusted: STRUCT //Is set by ASW
//      LN: UDT21210; //32 Bit
//      HN: UDT21210; //32 Bit 
//    END_STRUCT ;
//    InEnable: STRUCT // Target Pattern for BKT
//      LN: UDT21210; //32 Bit
//      HN: UDT21210; //32 Bit
//    END_STRUCT ;
//    OutEnable: STRUCT //Active way pattern 
//      LN: UDT21210; //32 Bit
//      HN: UDT21210; //32 Bit
//    END_STRUCT ;
//    InIsFlap   : UDT21210; //Changing immediately //16 Bit
//  END_STRUCT ;
//
//
// ------------------------------------------------------------
// Sequence Way change:
// ------------------------------------------------------------
// 1. Flaps of new way are adusted
// 2. Slide are opening
// 3. Add time is running
// 4. Slide are closing
//  
// 
//
//
AUTHOR : EA
FAMILY : GCS7LL
NAME : AddWay
VERSION : 4.4
VAR_INPUT
  InRcvCode : INT ;	//Gr.InCode
  InPointerPattern : ANY ;
  InModePassive : BOOL ;	//Gr.ModePassive
  InVarFault : BOOL ;	//Gr.VarFault
  InHoldOldWay : BOOL ;	//Do not activate the new pattern
  InAddTime : INT ;
  InAdjustTime : INT ;
  InBlowLine : BOOL ;
  InBKT : BOOL ;
END_VAR
VAR
  InStopAddTime : BOOL ;
  CmdImmediatelyChange : BOOL ;	//Change without adding time
  InElse : BOOL ;	//Active receiver is next group (only for BKT)
  Spare3 : BOOL ;
  Spare4 : BOOL ;
  Spare5 : BOOL ;
  Spare6 : BOOL ;
  Spare7 : BOOL ;
  CmdNewWay : BOOL ;	//Output: Pattern has changed
  OutAdjusted : BOOL ;	//All selected element are in the target position
  OutSlideAdjusted : BOOL ;	//All selected Slide gate adjusted
  OutFlapsAdjusted : BOOL ;	//All Selected Flaps are adjusted
  OutOldWayOK : BOOL ;	//During way change the old way is still ok
  OutNewWayOK : BOOL ;	//During way change the new way is still ok
  Spare216 : BOOL ;
  OutEnablePrev : BOOL ;	//Enable previous element
  OutConfigFault : BOOL ;	//Configuration fault pointer
  OutNewWayIsLonger : BOOL ;	//New Way Is Longer (command is only one scan high)
  OutNewWayIsShorter : BOOL ;	//New Way Is shorter (command is only one scan high)
  OutAdjustTimeRunning : BOOL ;	//Way adjust time running
  Spare224 : BOOL ;
  Spare225 : BOOL ;
  Spare226 : BOOL ;
  OutWayChangeActive : BOOL ;	//Old and new way pattern are added
  Internal : STRUCT
   OutModePassive : BOOL ;	//Is used for negative edge of ModePassive
   OutAddTimeRunning : BOOL ;	//old and new way pattern are active
   FlagElse : BOOL ;	//Positive edge of InElse
   Spare1 : BOOL ;
   Spare2 : BOOL ;
  END_STRUCT ;
  PatternOld : STRUCT
   InRcvCode : INT ;
   Position : INT ;	//Position Way Pattern
   EnableLN : DWORD ;
   EnableHN : DWORD ;
  END_STRUCT ;
  PatternNew : STRUCT 	//Is used to  detect change if the InEnableXxx
   InRcvCode : INT ;
   Position : INT ;	//Position Way Pattern
   EnableLN : DWORD ;
   EnableHN : DWORD ;
  END_STRUCT ;
  OutAddTime : INT ;
  OutAdjustTime : INT ;
  OutClosing : DWORD ;	//Slide gate must close
END_VAR
VAR_TEMP
  tmpWay_InAdjustedLN : DWORD ;	//Way.InAdjustedLN  Must be ar LD0 !!
  tmpWay_InAdjustedHN : DWORD ;	//Way.InAdjustedHN  Must be ar LD4 !!
  tmpWay_IsWayFlap : DWORD ;	//Way.InIsWayFlap   Must be at LD8 !!
  tmpEnableLN : DWORD ;	//Way.InAdjustedLN  Must be ar LD12 !!
  tmpEnableHN : DWORD ;	//Way.InAdjustedLN  Must be ar LD16 !!
  tmpWay_InEnableLN : DWORD ;	//Way.InEnableLN    Must be ar LD20 !!
  tmpWay_InEnableHN : DWORD ;	//Way.InEnableHN    Must be ar LD24 !!
  TmpOldSelectedWay : DWORD ;
  TmpNewSelectedWay : DWORD ;
  TmpReleaseChangeWay : DWORD ;
  TmpOldAndNewSelectedWay : DWORD ;
  tmp2ndLoop : BOOL ;
  tmpPatternArrayLen : INT ;
  tmpPatternArrayDB : INT ;
  tmpPatternArrayAddr : DWORD ;
  tmpPatternArrayEnd : DWORD ;	//End Address
  tmpAddrRead : DWORD ;
  tmpWay_OutEnableLN : DWORD ;	//Way.OutEnableLN
  tmpWay_OutEnableHN : DWORD ;	//Way.OutEnableHN
  tmpValue1 : DWORD ;
  tmpEnableFlaps : DWORD ;
  tmpEnableSlides : DWORD ;
  tmpSlideGates : DWORD ;
  tmpCnt : INT ;
  tmpAdjustedTempWay : BOOL ;	//Temporary way is adjusted
  tmpFlapsAdjusted : BOOL ;	//Flaps of temporary way is adjusted
  tmpFlapsOK : BOOL ;
  tmpSlidesOK : BOOL ;
  tmpSlideAdjustedHN : BOOL ;	//Slide of temporary way is adjusted (Aspiration flaps)
  tmpStoreEnableHN : DWORD ;
  tmpEmptyPattern : BOOL ;
END_VAR
BEGIN
NETWORK
TITLE = Calculate address of PatternArray
      L     P##InPointerPattern;
      L     W#16#FFFF;
      AD;
      LAR1  AR2;
      +AR1;	//--> Pointer to InPointerPattern
      L     DIW [AR1,P#0.0];
      L     DIW [AR1,P#4.0];
      T     #tmpPatternArrayDB;
      L     DID [AR1,P#6.0];
      T     #tmpPatternArrayAddr;
      L     DIW [AR1,P#2.0];
      L     26;
      <I;
      =     #OutConfigFault;
      R     #OutAdjusted;
      BEC;
NETWORK
TITLE = Load Pattern InAdjusted
      LAR1  #tmpPatternArrayAddr;
      L     DID [AR1,P#0.0];	// InAdjusted.LN
      T     #tmpWay_InAdjustedLN;
      L     DID [AR1,P#4.0];	// InAdjusted.HN
      T     #tmpWay_InAdjustedHN;
NETWORK
TITLE = Load Pattern InEnable
      +AR1  P#8.0;
      L     DID [AR1,P#0.0];	// InEnable.LN
      T     #tmpWay_InEnableLN;
      L     DID [AR1,P#4.0];	// InEnable.HN
      T     #tmpWay_InEnableHN;
      L     #tmpWay_InEnableLN;	//[4.1]
      L     #tmpWay_InEnableHN;	//[4.1]
      OD;	//[4.1]
      L     0;	//[4.1]
      ==D;	//[4.1]
      =     #tmpEmptyPattern;	//[4.1]   
NETWORK
TITLE = Load Pattern OutEnable
      +AR1  P#8.0;
      L     DID [AR1,P#0.0];	// OutEnable.LN
      T     #tmpWay_OutEnableLN;
      L     DID [AR1,P#4.0];	// OutEnable.HN
      T     #tmpWay_OutEnableHN;
      T     #tmpStoreEnableHN;
NETWORK
TITLE = Load Pattern InIsWayFlap
      +AR1  P#8.0;
      L     DID [AR1,P#0.0];	// InIsWayFlap
      T     #tmpWay_IsWayFlap;
      INVD;
      T     #tmpSlideGates;
NETWORK
TITLE = Init Flag Part 1:
      CLR;
      =     #OutNewWayIsLonger;
      =     #OutNewWayIsShorter;
NETWORK
TITLE = Hold Old Pattern, if inCode is not ok
      A     #InElse;
      FP    #Internal.FlagElse;
      O     #InHoldOldWay;
      JCN   HOJ0;
      L     #PatternNew.EnableLN;
      T     #tmpWay_InEnableLN;
      L     #PatternNew.EnableHN;
      T     #tmpWay_InEnableHN;
HOJ0: NOP   0;
NETWORK
TITLE = Test if target position has changed
      A(;
      L     #PatternNew.EnableLN;
      L     #tmpWay_InEnableLN;
      <>D;
      );
      O(;
      L     #PatternNew.EnableHN;
      L     #tmpWay_InEnableHN;
      <>D;
      );
      =     #CmdNewWay;
      A     #CmdNewWay;
      JCN   AD10;
//-->Store new Pattern in PatternNew
      L     #InRcvCode;
      T     #PatternNew.InRcvCode;
      L     #tmpWay_InEnableLN;
      T     #PatternNew.EnableLN;
      L     #tmpWay_InEnableHN;
      T     #PatternNew.EnableHN;
      L     #InAddTime;
      T     #OutAddTime;
//====================================
//Calculate position
//-------------------
//Search last bit in PatternNew.EnableHN
//For flaps use LN or HN
      A     #InElse;
      L     33;
      JC    AD9;
      L     #tmpWay_InEnableLN;
      L     #tmpWay_InEnableHN;
      OD;
      L     #tmpWay_IsWayFlap;
      AD;
//For Slides use only HN
      L     #tmpWay_InEnableHN;
      OD;
      CAD;
      T     #tmpValue1;
      L     32;
ADLO: T     #PatternNew.Position;
      L     #tmpValue1;
      SRD   1;
      JP    AD10;
      T     #tmpValue1;
      L     #PatternNew.Position;
      LOOP  ADLO;
      L     0;
AD9:  T     #PatternNew.Position;
AD10: NOP   0;
NETWORK
TITLE = Test is way is long
      L     #PatternNew.Position;
      L     #PatternOld.Position;
      >I;
      O     #InElse;
      A     #InBKT;	//[4.2]
      =     #OutNewWayIsLonger;
      <I;
      AN    #InElse;
      A     #InBKT;	//[4.2]
      =     #OutNewWayIsShorter;
NETWORK
TITLE = Compare InEnableXxx with OutEnableXxx
      L     #tmpWay_InEnableLN;
      L     #tmpWay_OutEnableLN;
      <>D;
      O(;
      L     #tmpWay_InEnableHN;
      L     #tmpWay_OutEnableHN;
      <>D;
      );
      FN    #OutWayChangeActive;
      S     #CmdNewWay;	//[4.4]
NETWORK
TITLE = Add Old way and way of new selected elements
////------------------------------------------------------------------------
////CASE: Add only new selected element, hold way of old selected elements    
////------------------------------------------------------------------------
      AN    #OutWayChangeActive;
      O     #CmdNewWay;
      JC    ADN0;
//Select new element
      L     #tmpWay_OutEnableLN;
      L     #tmpWay_OutEnableHN;
      OD;
      T     #TmpOldSelectedWay;
      L     #PatternNew.EnableLN;
      L     #PatternNew.EnableHN;
      OD;
      T     #TmpNewSelectedWay;
      L     #TmpOldSelectedWay;
      L     #TmpNewSelectedWay;
      AD;
      T     #TmpOldAndNewSelectedWay;
      L     #tmpWay_OutEnableLN;
      L     #PatternNew.EnableLN;
      XOD;
      L     #TmpOldAndNewSelectedWay;
      AD;
      INVD;
      T     #TmpReleaseChangeWay;	//<<--- OLD+NEW+CHANGE 
      AN    #InBKT;	//[4.3]
      O     #InHoldOldWay;	//[4.3]
      JC    AD43;	//[4.3]
      L     #TmpReleaseChangeWay;	//[4.3]
      L     #tmpWay_IsWayFlap;	//[4.3]
      OD;	//[4.3]
      T     #TmpReleaseChangeWay;	//<<--- OLD+NEW+CHANGE 
AD43: NOP   0;
//--> Set Bits in  tmpWay_OutEnableHN 
      L     #PatternNew.EnableHN;
      L     #TmpReleaseChangeWay;
      AD;
      L     #tmpWay_OutEnableHN;
      OD;
      T     #tmpWay_OutEnableHN;
//--> Reset Bits in  tmpWay_OutEnableLN 
      INVD;
      L     #tmpWay_OutEnableLN;
      AD;
      T     #tmpWay_OutEnableLN;
//--> Set Bits in  tmpWay_OutEnableLN 
      L     #PatternNew.EnableLN;
      L     #TmpReleaseChangeWay;
      AD;
      L     #tmpWay_OutEnableLN;
      OD;
      T     #tmpWay_OutEnableLN;
//--> Reset Bits in  tmpWay_OutEnableHN
      INVD;
      L     #tmpWay_OutEnableHN;
      AD;
      T     #tmpWay_OutEnableHN;
ADN0: NOP   0;
NETWORK
TITLE = Test Flaps Adjusted
      AN    #OutWayChangeActive;
      JC    AJF1;
      A(;
      L     #tmpWay_OutEnableLN;
      L     #tmpWay_IsWayFlap;
      AD;
      T     #tmpEnableFlaps;
      L     #tmpWay_InAdjustedLN;
      AD;
      L     #tmpEnableFlaps;
      ==D;
      );
      A(;
      L     #tmpWay_OutEnableHN;
      L     #tmpWay_IsWayFlap;
      AD;
      T     #tmpEnableFlaps;
      L     #tmpWay_InAdjustedHN;
      AD;
      L     #tmpEnableFlaps;
      ==D;
      );
AJF1: A     #OutWayChangeActive;
      =     #tmpFlapsAdjusted;
NETWORK
TITLE = Add EnableHN of Slide Gate of old and new way 
      AN    #tmpFlapsAdjusted;
      AN    #InBlowLine;
      ON    #OutWayChangeActive;
      O     #CmdNewWay;
      JC    ADJ0;
//--> Set Bits in  tmpWay_OutEnableHN 
      AN    #OutNewWayOK;
      O     #Internal.OutAddTimeRunning;
      JC    ADJ1;
//Old flap not langer in st HN            //[3.1 -->
      L     #PatternOld.EnableHN;
      L     #PatternNew.EnableHN;
      INVD;
      AD;
      L     #tmpSlideGates;
      AD;	//Not used in new pattern
      L     #tmpWay_InAdjustedHN;
      INVD;
      AD;	// flap has change from StHN --> StLN
      INVD;
      L     #tmpWay_OutEnableHN;
      AD;
      T     #tmpWay_OutEnableHN;	//<-- 3.1]
ADJ1: L     #PatternNew.EnableHN;
      L     #tmpSlideGates;
      AD;
      L     #tmpWay_OutEnableHN;
      OD;
      T     #tmpWay_OutEnableHN;
//--> Reset Bits in  tmpWay_OutEnableLN 
      INVD;
      L     #tmpWay_OutEnableLN;
      AD;
      T     #tmpWay_OutEnableLN;
ADJ0: NOP   0;
NETWORK
TITLE = Run Add Time
      AN    #OutWayChangeActive;
      JC    TAJ0;
//delay time
      A     "GCS7_Gr_OutTick200ms";
      AN    #InStopAddTime;
      A(;
      L     #OutAddTime;
      L     0;
      >I;
      );
      JCN   TAJ1;
      L     #OutAddTime;
      +     -2;
      T     #OutAddTime;
TAJ1: L     #OutAddTime;
      L     0;
      >I;
TAJ0: A     #OutWayChangeActive;
      =     #Internal.OutAddTimeRunning;
NETWORK
TITLE = Test added way is adjusted
//All elements of the actual pattern are in adjusted
      AN    #OutWayChangeActive;
      JC    TAO1;
      L     #tmpWay_InAdjustedLN;
      L     #tmpWay_OutEnableLN;
      AD;
      L     #tmpWay_OutEnableLN;
      ==D;
      A(;
      L     #tmpWay_InAdjustedHN;
      L     #tmpWay_OutEnableHN;
      AD;
      L     #tmpWay_OutEnableHN;
      ==D;
      );
TAO1: A     #OutWayChangeActive;
      =     #tmpAdjustedTempWay;
NETWORK
TITLE = Change Old Way Flap of Blow Line
//The old way flaps are changed if the aspiration flaps and the new way elements 
//are adjusted
      AN    #OutWayChangeActive;
      JC    OFJ0;
      AN    #InBlowLine;
      ON    #tmpAdjustedTempWay;
      O     #CmdNewWay;
      JC    OFJ0;
//--> Set Bits in  tmpWay_OutEnableHN 
      L     #PatternNew.EnableHN;
      L     #tmpWay_IsWayFlap;
      AD;
      L     #tmpWay_OutEnableHN;
      OD;
      T     #tmpWay_OutEnableHN;
//--> Reset Bits in  tmpWay_OutEnableLN 
      INVD;
      L     #tmpWay_OutEnableLN;
      AD;
      T     #tmpWay_OutEnableLN;
//--> Set Bits in  tmpWay_OutEnableLN 
      L     #PatternNew.EnableLN;
      L     #tmpWay_IsWayFlap;
      AD;
      L     #tmpWay_OutEnableLN;
      OD;
      T     #tmpWay_OutEnableLN;
//--> Reset Bits in  tmpWay_OutEnableHN
      INVD;
      L     #tmpWay_OutEnableHN;
      AD;
      T     #tmpWay_OutEnableHN;
OFJ0: NOP   0;
NETWORK
TITLE = CmdNewWay (Case 2)
      LAR1  #tmpPatternArrayAddr;
      +AR1  P#16.0;
      L     #tmpWay_OutEnableLN;
      L     DID [AR1,P#0.0];	//Way.OutEnable.LN
      <>D;
      O(;
      L     #tmpStoreEnableHN;	//[4.3] #tmpWay_OutEnableHN
      L     DID [AR1,P#4.0];	//Way.OutEnable.HN
      <>D;
      );
      S     #CmdNewWay;
NETWORK
TITLE = Activate new way pattern
//=======================
//ModePassive or Transition ModePassive--> ModeActive
      A     #InModePassive;
      FN    #Internal.OutModePassive;
      O     #InModePassive;
      JC    AWN1;
//=======================
      AN    #Internal.OutAddTimeRunning;
      O     #CmdImmediatelyChange;
      AN    #CmdNewWay;
      A(;
      O     #tmpAdjustedTempWay;
      O     #OutAdjusted;
      O;
      A     #InVarFault;
      A     #CmdImmediatelyChange;
      );
      JCN   AWN0;
//=======================
//Copy Pattern
AWN1: L     #PatternNew.EnableLN;
      T     #tmpWay_OutEnableLN;	//Way.OutEnable.LN
      L     #PatternNew.EnableHN;
      T     #tmpWay_OutEnableHN;	//Way.OutEnable.HN
//Copy new pattern to old pattern
      AN    #OutAdjusted;
      JC    AWN0;
      L     #PatternNew.InRcvCode;
      T     #PatternOld.InRcvCode;
      L     #PatternNew.EnableLN;
      T     #PatternOld.EnableLN;
      L     #PatternNew.EnableHN;
      T     #PatternOld.EnableHN;
      L     #PatternNew.Position;
      T     #PatternOld.Position;
      R     #OutWayChangeActive;
AWN0: NOP   0;
NETWORK
TITLE = Test Adjusted =  OutAdjusted
      L     #tmpWay_InAdjustedLN;
      L     #tmpWay_InEnableLN;
      AD;
      L     #tmpWay_InEnableLN;
      ==D;
      A(;
      L     #tmpWay_InAdjustedHN;
      L     #tmpWay_InEnableHN;
      AD;
      L     #tmpWay_InEnableHN;
      ==D;
      );
      AN    #InHoldOldWay;
      AN    #tmpEmptyPattern;	//[4.1] 
      =     #OutAdjusted;
NETWORK
TITLE = Run OutAdjustTime
      AN    #CmdNewWay;
      JC    ATJ2;
//==================================
//Start Adjust Time
      L     #InAdjustTime;
      T     #OutAdjustTime;
//=================================
//Run Adjust Time
ATJ2: A     "GCS7_Gr_OutTick200ms";
      A(;
      L     #OutAdjustTime;
      L     0;
      >I;
      );
      JCN   ATJ3;
      L     #OutAdjustTime;
      +     -2;
      T     #OutAdjustTime;
ATJ3: L     #OutAdjustTime;
      L     0;
      >I;
      =     #OutAdjustTimeRunning;
NETWORK
TITLE = Test Flaps Adjusted
//Is used during way change to test if still a way is ok
      A     #OutAdjusted;
      JC    AFJ0;
      L     #tmpWay_OutEnableLN;
      L     #tmpWay_IsWayFlap;
      AD;
      T     #tmpEnableFlaps;
      L     #tmpWay_InAdjustedLN;
      AD;
      L     #tmpEnableFlaps;
      ==D;
      A(;
      L     #tmpWay_OutEnableHN;
      L     #tmpWay_IsWayFlap;
      AD;
      T     #tmpEnableFlaps;
      L     #tmpWay_InAdjustedHN;
      AD;
      L     #tmpEnableFlaps;
      ==D;
      );
AFJ0: =     #OutFlapsAdjusted;
NETWORK
TITLE = Test Slide Adjusted
//Is used during way change to test if still a way is ok
      A     #OutAdjusted;
      JC    ASJ0;
      L     #tmpWay_OutEnableLN;
      L     #tmpSlideGates;
      AD;
      T     #tmpEnableSlides;
      L     #tmpWay_InAdjustedLN;
      AD;
      L     #tmpEnableSlides;
      ==D;
      A(;
      L     #tmpWay_OutEnableHN;
      L     #tmpSlideGates;
      AD;
      T     #tmpEnableSlides;
      L     #tmpWay_InAdjustedHN;
      AD;
      L     #tmpEnableSlides;
      ==D;
      );
ASJ0: =     #OutSlideAdjusted;
NETWORK
TITLE = Test Old Way still ok
//Condition:
// 1. All Slides are in target postion
// 2. All Flaps of the old way are in target position
//
//Thsi function works because the flaps are always first ajusted 
      A     #OutAdjusted;
      R     #OutOldWayOK;
      JC    WOJ0;
//=======================================================
//CASE1: IF all Slides are adjusted check only the flaps
//=======================================================
      AN    #OutSlideAdjusted;
      JC    WOSL;
//Test Flaps adjusted 
      L     #PatternOld.EnableLN;
      L     #tmpWay_IsWayFlap;
      AD;
      T     #tmpEnableFlaps;
      L     #tmpWay_InAdjustedLN;
      AD;
      L     #tmpEnableFlaps;
      ==D;
      A(;
      L     #PatternOld.EnableHN;
      L     #tmpWay_IsWayFlap;
      AD;
      T     #tmpEnableFlaps;
      L     #tmpWay_InAdjustedHN;
      AD;
      L     #tmpEnableFlaps;
      ==D;
      );
      A     #OutSlideAdjusted;
      =     #OutOldWayOK;
      JU    WOJ0;
//=======================================================
//CASE: All flaps are adjusted: New Slides not relevant for closed
//=======================================================
WOSL: L     #PatternOld.EnableLN;
      L     #tmpWay_InEnableHN;	//--> New Slides not relevant for closed
      INVD;
      AD;
      L     #tmpSlideGates;
      AD;
      T     #tmpEnableSlides;
      L     #tmpWay_InAdjustedLN;
      AD;
      L     #tmpEnableSlides;
      ==D;
      A(;
      L     #PatternOld.EnableHN;
      L     #tmpSlideGates;
      AD;
      T     #tmpEnableSlides;
      L     #tmpWay_InAdjustedHN;
      AD;
      L     #tmpEnableSlides;
      ==D;
      );
      =     #tmpSlidesOK;
      A     #tmpSlidesOK;
      A     #OutFlapsAdjusted;
      =     #OutOldWayOK;
WOJ0: NOP   0;
      L     #PatternOld.EnableLN;	//[4.1]
      L     #PatternOld.EnableHN;	//[4.1]
      OD;	//[4.1]
      L     0;	//[4.1]
      ==D;	//[4.1]
      R     #OutOldWayOK;	//[4.1]
NETWORK
TITLE = Test New Way ok
//Condition:
// 1. All Slides are in target postion
// 2. All Flaps of the new way are in target position
//
//Thsi function works because the flaps are always first ajusted 
      A     #OutAdjusted;
      S     #OutNewWayOK;
      JC    WNJ0;
//Detect closing command
      L     #tmpStoreEnableHN;
      L     #tmpWay_OutEnableLN;
      AD;
      L     #tmpSlideGates;
      AD;
      L     #OutClosing;
      OD;
      L     #tmpWay_OutEnableHN;
      INVD;
      AD;
      L     #tmpWay_InAdjustedLN;
      INVD;
      AD;
      T     #OutClosing;
//=======================================================
//CASE1: IF all Slides are adjusted check only the flaps
//=======================================================
      AN    #OutSlideAdjusted;
      JC    WNSL;
      L     #tmpWay_InEnableLN;
      L     #tmpWay_IsWayFlap;
      AD;
      T     #tmpEnableFlaps;
      L     #tmpWay_InAdjustedLN;
      AD;
      L     #tmpEnableFlaps;
      ==D;
      A(;
      L     #tmpWay_InEnableHN;
      L     #tmpWay_IsWayFlap;
      AD;
      T     #tmpEnableFlaps;
      L     #tmpWay_InAdjustedHN;
      AD;
      L     #tmpEnableFlaps;
      ==D;
      );
      A     #OutSlideAdjusted;
      AN    #tmpEmptyPattern;	//[4.1] 
      =     #OutNewWayOK;
      JU    WNJ0;
//=======================================================
//CASE: All flaps are adjusted: Old Slides not relevant for close
//=======================================================
WNSL: L     #tmpWay_InEnableLN;
      L     #PatternOld.EnableHN;	//--> New Slide not relevant for closed
      INVD;
      AD;
      L     #tmpSlideGates;
      AD;
      T     #tmpEnableSlides;
      L     #tmpEnableSlides;
      L     #OutClosing;	//[2.0] Closing slide are not relevant for closed
      AD;
      L     #tmpWay_InAdjustedLN;
      OD;
      L     #tmpEnableSlides;
      AD;
      L     #tmpEnableSlides;
      ==D;
      A(;
      L     #tmpWay_InEnableHN;
      L     #tmpSlideGates;
      AD;
      T     #tmpEnableSlides;
      L     #tmpWay_InAdjustedHN;
      AD;
      L     #tmpEnableSlides;
      ==D;
      );
      AN    #OutSlideAdjusted;
      =     #tmpSlidesOK;
      A     #tmpSlidesOK;
      A     #OutFlapsAdjusted;
      AN    #tmpEmptyPattern;	//[4.1] 
      =     #OutNewWayOK;
WNJ0: NOP   0;
NETWORK
TITLE =
      AN    #OutEnablePrev;
      O     #OutAdjusted;
      O     #InVarFault;
      JCN   CLOS;
      L     0;
      T     #OutClosing;
CLOS: NOP   0;
NETWORK
TITLE = BKT:  [4.0]
//Problem: 
//When changing 3 time, then during add time perhaps 3 slide gates are open.
// Longer way --> shorter way --> position between 
//Solution:
//  Reset OutEnableHN of slide gate in shorter way then the new way
      AN    #InBKT;
      JC    BKJ0;
      AN    #OutNewWayOK;
      O     #OutAdjusted;
      ON    #OutFlapsAdjusted;
      JC    BKJ0;
      L     #PatternNew.Position;
      L     #PatternOld.Position;
      >I;
      JC    BKJ0;
//==================================================
//Test new Slide gates are open
//--------------------------------------------------
      A(;
      L     #tmpWay_InAdjustedHN;
      L     #tmpWay_InEnableHN;
      AD;
      L     #tmpWay_InEnableHN;
      ==D;
      );
      AN    #InHoldOldWay;
      JCN   BKJ0;
//==================================================
//Calculate Pattern for shorter way then the new way
//--------------------------------------------------
      L     33;
      L     #PatternNew.Position;
      -D;
      T     #tmpCnt;
      L     DW#16#FFFFFFFF;
      SLD;
      INVD;
      L     #tmpWay_IsWayFlap;	//Not used for flap
      CAD;
      OD;
//==================================================
//Reset OutEnableHN of slide gate in shorter way 
//==================================================
      L     #tmpWay_OutEnableHN;
      CAD;
      AD;
      CAD;
      T     #tmpWay_OutEnableHN;
BKJ0: NOP   0;
NETWORK
TITLE = OutEnableNext
      A     #OutAdjustTimeRunning;
      A     #OutEnablePrev;
      O     #OutOldWayOK;
      O     #OutNewWayOK;
      O     #OutAdjusted;
//      UN    #InHoldOldWay
      =     #OutEnablePrev;
NETWORK
TITLE = Store Output Data: 
      LAR1  #tmpPatternArrayAddr;
      +AR1  P#16.0;
      L     #tmpWay_OutEnableLN;
      T     DID [AR1,P#0.0];	//Way.OutEnable.LN
      L     #tmpWay_OutEnableHN;
      T     DID [AR1,P#4.0];	//Way.OutEnable.HN
//Init Flag
      SET;
      R     #CmdImmediatelyChange;
END_FUNCTION_BLOCK

